LIN {X 0,Y 404.076,Z 442.331,A -85,B 0,C 180,E1 -11324.748,E2 -11324.748} C_VEL
LIN {X 0,Y 402.953,Z 452.471,A -85,B 0,C 180,E1 -11326.125,E2 -11326.125} C_VEL
LIN {X 0,Y 401.871,Z 461.516,A -85,B 0,C 180,E1 -11327.63,E2 -11327.63} C_VEL
LIN {X 0,Y 400.856,Z 469.336,A -85,B 0,C 180,E1 -11329.213,E2 -11329.213} C_VEL
LIN {X 0,Y 399.877,Z 476.001,A -85,B 0,C 180,E1 -11330.899,E2 -11330.899} C_VEL
LIN {X 0,Y 399.254,Z 480.643,A -85,B 0,C 180,E1 -11332.414,E2 -11332.414} C_VEL
LIN {X 0,Y 398.694,Z 484.232,A -85,B 0,C 180,E1 -11333.929,E2 -11333.929} C_VEL
LIN {X 0,Y 398.541,Z 486.049,A -85,B 0,C 180,E1 -11334.942,E2 -11334.942} C_VEL
LIN {X 0,Y 398.272,Z 487.43,A -85,B 0,C 180,E1 -11335.953,E2 -11335.953} C_VEL
LIN {X 0,Y 398.06,Z 488.39,A -85,B 0,C 180,E1 -11336.964,E2 -11336.964} C_VEL
LIN {X 0,Y 397.79,Z 488.969,A -85,B 0,C 180,E1 -11337.975,E2 -11337.975} C_VEL
LIN {X 0,Y 397.658,Z 489.133,A -85,B 0,C 180,E1 -11338.988,E2 -11338.988} C_VEL
LIN {X 0,Y 397.526,Z 488.893,A -85,B 0,C 180,E1 -11340,E2 -11340} C_VEL
LIN {X 0,Y 397.495,Z 488.205,A -85,B 0,C 180,E1 -11341.013,E2 -11341.013} C_VEL
LIN {X 0,Y 397.414,Z 487.123,A -85,B 0,C 180,E1 -11342.027,E2 -11342.027} C_VEL
LIN {X 0,Y 397.512,Z 485.612,A -85,B 0,C 180,E1 -11343.041,E2 -11343.041} C_VEL
LIN {X 0,Y 397.477,Z 482.566,A -85,B 0,C 180,E1 -11344.564,E2 -11344.564} C_VEL
LIN {X 0,Y 397.578,Z 478.489,A -85,B 0,C 180,E1 -11346.089,E2 -11346.089} C_VEL
LIN {X 0,Y 398.065,Z 473.274,A -85,B 0,C 180,E1 -11347.61,E2 -11347.61} C_VEL
LIN {X 0,Y 398.488,Z 465.684,A -85,B 0,C 180,E1 -11349.39,E2 -11349.39} C_VEL
LIN {X 0,Y 398.962,Z 457.56,A -85,B 0,C 180,E1 -11350.916,E2 -11350.916} C_VEL
LIN {X 0,Y 399.517,Z 447.676,A -85,B 0,C 180,E1 -11352.445,E2 -11352.445} C_VEL
LIN {X 0,Y 400.278,Z 437.712,A -85,B 0,C 180,E1 -11353.712,E2 -11353.712} C_VEL
LIN {X 0,Y 400.99,Z 425.569,A -85,B 0,C 180,E1 -11354.983,E2 -11354.983} C_VEL
LIN {X 0,Y 401.633,Z 413.729,A -85,B 0,C 180,E1 -11355.995,E2 -11355.995} C_VEL
LIN {X 0,Y 402.443,Z 400.813,A -85,B 0,C 180,E1 -11356.878,E2 -11356.878} C_VEL
LIN {X 0,Y 402.734,Z 392.913,A -85,B 0,C 180,E1 -11357.323,E2 -11357.323} C_VEL
LIN {X 0,Y 399.412,Z 378.284,A -85,B 0,C 180,E1 -11358.158,E2 -11358.158} C_VEL
LIN {X 0,Y 396.905,Z 368.546,A -85,B 0,C 180,E1 -11358.62,E2 -11358.62} C_VEL
LIN {X 0,Y 397.081,Z 362.565,A -85,B 0,C 180,E1 -11361.82,E2 -11361.82} C_VEL
LIN {X 0,Y 397.308,Z 355.709,A -85,B 0,C 180,E1 -11365.556,E2 -11365.556} C_VEL
LIN {X 0,Y 397.543,Z 349.381,A -85,B 0,C 180,E1 -11369.089,E2 -11369.089} C_VEL
LIN {X 0,Y 397.831,Z 343.175,A -85,B 0,C 180,E1 -11372.603,E2 -11372.603} C_VEL
LIN {X 0,Y 397.935,Z 337.889,A -85,B 0,C 180,E1 -11375.665,E2 -11375.665} C_VEL
LIN {X 0,Y 397.733,Z 335.123,A -85,B 0,C 180,E1 -11377.328,E2 -11377.328} C_VEL
LIN {X 0,Y 397.121,Z 331.336,A -85,B 0,C 180,E1 -11379.735,E2 -11379.735} C_VEL
LIN {X 0,Y 397.109,Z 331.334,A -85,B 0,C 180,E1 -11383.648,E2 -11383.648} C_VEL
LIN {X 0,Y 397.11,Z 331.332,A -85,B 0,C 180,E1 -11386.52,E2 -11386.52} C_VEL
LIN {X 0,Y 397.128,Z 331.421,A -85,B 0,C 180,E1 -11390.027,E2 -11390.027} C_VEL
LIN {X 0,Y 398.424,Z 338.477,A -85,B 0,C 180,E1 -11393.146,E2 -11393.146} C_VEL
LIN {X 0,Y 398.848,Z 342.731,A -85,B 0,C 180,E1 -11395.061,E2 -11395.061} C_VEL
LIN {X 0,Y 398.687,Z 350.568,A -85,B 0,C 180,E1 -11398.664,E2 -11398.664} C_VEL
LIN {X 0,Y 398.55,Z 357.361,A -85,B 0,C 180,E1 -11401.848,E2 -11401.848} C_VEL
LIN {X 0,Y 398.521,Z 365.236,A -85,B 0,C 180,E1 -11405.515,E2 -11405.515} C_VEL
LIN {X 0,Y 398.622,Z 373.552,A -85,B 0,C 180,E1 -11409.137,E2 -11409.137} C_VEL
LIN {X 0,Y 398.818,Z 380.793,A -85,B 0,C 180,E1 -11411.941,E2 -11411.941} C_VEL
LIN {X 0,Y 402.682,Z 393.199,A -85,B 0,C 180,E1 -11412.494,E2 -11412.494} C_VEL
LIN {X 0,Y 403.209,Z 396.027,A -85,B 0,C 180,E1 -11412.631,E2 -11412.631} C_VEL
LIN {X 0,Y 402.908,Z 408.015,A -85,B 0,C 180,E1 -11413.206,E2 -11413.206} C_VEL
LIN {X 0,Y 402.433,Z 419.434,A -85,B 0,C 180,E1 -11413.95,E2 -11413.95} C_VEL
LIN {X 0,Y 401.82,Z 430.918,A -85,B 0,C 180,E1 -11414.918,E2 -11414.918} C_VEL
LIN {X 0,Y 401.129,Z 441.593,A -85,B 0,C 180,E1 -11416.058,E2 -11416.058} C_VEL
LIN {X 0,Y 400.428,Z 451.077,A -85,B 0,C 180,E1 -11417.325,E2 -11417.325} C_VEL
LIN {X 0,Y 399.552,Z 460.293,A -85,B 0,C 180,E1 -11418.841,E2 -11418.841} C_VEL
LIN {X 0,Y 398.974,Z 467.575,A -85,B 0,C 180,E1 -11420.365,E2 -11420.365} C_VEL
LIN {X 0,Y 398.52,Z 473.405,A -85,B 0,C 180,E1 -11421.887,E2 -11421.887} C_VEL
LIN {X 0,Y 397.835,Z 478.062,A -85,B 0,C 180,E1 -11423.404,E2 -11423.404} C_VEL
LIN {X 0,Y 397.571,Z 481.583,A -85,B 0,C 180,E1 -11424.927,E2 -11424.927} C_VEL
LIN {X 0,Y 397.535,Z 483.38,A -85,B 0,C 180,E1 -11425.943,E2 -11425.943} C_VEL
LIN {X 0,Y 397.447,Z 484.762,A -85,B 0,C 180,E1 -11426.957,E2 -11426.957} C_VEL
LIN {X 0,Y 397.196,Z 486.352,A -85,B 0,C 180,E1 -11428.984,E2 -11428.984} C_VEL
LIN {X 0,Y 397.16,Z 486.586,A -85,B 0,C 180,E1 -11429.998,E2 -11429.998} C_VEL
LIN {X 0,Y 397.293,Z 485.82,A -85,B 0,C 180,E1 -11432.025,E2 -11432.025} C_VEL
LIN {X 0,Y 397.459,Z 484.866,A -85,B 0,C 180,E1 -11433.038,E2 -11433.038} C_VEL
LIN {X 0,Y 397.552,Z 483.541,A -85,B 0,C 180,E1 -11434.052,E2 -11434.052} C_VEL
LIN {X 0,Y 397.722,Z 480.756,A -85,B 0,C 180,E1 -11435.575,E2 -11435.575} C_VEL
LIN {X 0,Y 398.1,Z 476.945,A -85,B 0,C 180,E1 -11437.096,E2 -11437.096} C_VEL
LIN {X 0,Y 398.64,Z 471.995,A -85,B 0,C 180,E1 -11438.616,E2 -11438.616} C_VEL
LIN {X 0,Y 398.848,Z 469.563,A -85,B 0,C 180,E1 -11439.249,E2 -11439.249} C_VEL
LIN {X 0,Y 398.363,Z 467.668,A -85,B 0,C 180,E1 -11439.75,E2 -11439.75} C_VEL
LIN {X 0,Y 393.286,Z 461.707,A -85,B 0,C 180,E1 -11441.349,E2 -11441.349} C_VEL
LIN {X 0,Y 392.936,Z 459.353,A -85,B 0,C 180,E1 -11441.816,E2 -11441.816} C_VEL
LIN {X 0,Y 393.736,Z 451.114,A -85,B 0,C 180,E1 -11443.152,E2 -11443.152} C_VEL
LIN {X 0,Y 394.369,Z 442.445,A -85,B 0,C 180,E1 -11444.313,E2 -11444.313} C_VEL
LIN {X 0,Y 395.042,Z 431.694,A -85,B 0,C 180,E1 -11445.474,E2 -11445.474} C_VEL
LIN {X 0,Y 395.736,Z 420.066,A -85,B 0,C 180,E1 -11446.462,E2 -11446.462} C_VEL
LIN {X 0,Y 396.267,Z 408.557,A -85,B 0,C 180,E1 -11447.212,E2 -11447.212} C_VEL
LIN {X 0,Y 396.362,Z 396.075,A -85,B 0,C 180,E1 -11447.817,E2 -11447.817} C_VEL
LIN {X 0,Y 392.761,Z 384.449,A -85,B 0,C 180,E1 -11448.381,E2 -11448.381} C_VEL
LIN {X 0,Y 391.906,Z 381.637,A -85,B 0,C 180,E1 -11448.505,E2 -11448.505} C_VEL
LIN {X 0,Y 391.687,Z 373.901,A -85,B 0,C 180,E1 -11451.578,E2 -11451.578} C_VEL
LIN {X 0,Y 391.648,Z 367.501,A -85,B 0,C 180,E1 -11454.373,E2 -11454.373} C_VEL
LIN {X 0,Y 391.635,Z 359.97,A -85,B 0,C 180,E1 -11457.809,E2 -11457.809} C_VEL
LIN {X 0,Y 391.769,Z 354.179,A -85,B 0,C 180,E1 -11460.561,E2 -11460.561} C_VEL
LIN {X 0,Y 391.906,Z 347.231,A -85,B 0,C 180,E1 -11463.77,E2 -11463.77} C_VEL
LIN {X 0,Y 391.796,Z 341.719,A -85,B 0,C 180,E1 -11466.292,E2 -11466.292} C_VEL
LIN {X 0,Y 390.605,Z 335.016,A -85,B 0,C 180,E1 -11469.314,E2 -11469.314} C_VEL
LIN {X 0,Y 390.047,Z 332.214,A -85,B 0,C 180,E1 -11470.531,E2 -11470.531} C_VEL
LIN {X 0,Y 390.044,Z 332.214,A -85,B 0,C 180,E1 -11473.884,E2 -11473.884} C_VEL
LIN {X 0,Y 390.099,Z 332.208,A -85,B 0,C 180,E1 -11476.795,E2 -11476.795} C_VEL
LIN {X 0,Y 390.063,Z 332.208,A -85,B 0,C 180,E1 -11479.561,E2 -11479.561} C_VEL
LIN {X 0,Y 390.031,Z 332.215,A -85,B 0,C 180,E1 -11482.446,E2 -11482.446} C_VEL
LIN {X 0,Y 390.05,Z 332.211,A -85,B 0,C 180,E1 -11486.043,E2 -11486.043} C_VEL
LIN {X 0,Y 390.027,Z 332.209,A -85,B 0,C 180,E1 -11489.867,E2 -11489.867} C_VEL
LIN {X 0,Y 390.093,Z 332.199,A -85,B 0,C 180,E1 -11493.23,E2 -11493.23} C_VEL
LIN {X 0,Y 390.102,Z 332.198,A -85,B 0,C 180,E1 -11496.743,E2 -11496.743} C_VEL
LIN {X 0,Y 390.108,Z 332.202,A -85,B 0,C 180,E1 -11499.983,E2 -11499.983} C_VEL
LIN {X 0,Y 390.115,Z 332.206,A -85,B 0,C 180,E1 -11503.247,E2 -11503.247} C_VEL
LIN {X 0,Y 390.171,Z 332.189,A -85,B 0,C 180,E1 -11506.56,E2 -11506.56} C_VEL
LIN {X 0,Y 390.159,Z 332.195,A -85,B 0,C 180,E1 -11509.622,E2 -11509.622} C_VEL
LIN {X 0,Y 390.294,Z 332.18,A -85,B 0,C 180,E1 -11512.758,E2 -11512.758} C_VEL
LIN {X 0,Y 390.203,Z 332.187,A -85,B 0,C 180,E1 -11514.833,E2 -11514.833} C_VEL
LIN {X 0,Y 390.392,Z 332.168,A -85,B 0,C 180,E1 -11517.936,E2 -11517.936} C_VEL
LIN {X 0,Y 390.524,Z 332.147,A -85,B 0,C 180,E1 -11520,E2 -11520} C_VEL
LIN {X 0,Y 390.328,Z 332.176,A -85,B 0,C 180,E1 -11523.096,E2 -11523.096} C_VEL
LIN {X 0,Y 390.317,Z 332.177,A -85,B 0,C 180,E1 -11526.202,E2 -11526.202} C_VEL
LIN {X 0,Y 390.29,Z 332.181,A -85,B 0,C 180,E1 -11528.282,E2 -11528.282} C_VEL
LIN {X 0,Y 390.154,Z 332.2,A -85,B 0,C 180,E1 -11532.483,E2 -11532.483} C_VEL
LIN {X 0,Y 390.12,Z 332.202,A -85,B 0,C 180,E1 -11535.677,E2 -11535.677} C_VEL
LIN {X 0,Y 390.097,Z 332.205,A -85,B 0,C 180,E1 -11538.922,E2 -11538.922} C_VEL
LIN {X 0,Y 390.09,Z 332.206,A -85,B 0,C 180,E1 -11542.231,E2 -11542.231} C_VEL
LIN {X 0,Y 390.096,Z 332.204,A -85,B 0,C 180,E1 -11545.745,E2 -11545.745} C_VEL
LIN {X 0,Y 390.036,Z 332.212,A -85,B 0,C 180,E1 -11549.111,E2 -11549.111} C_VEL
LIN {X 0,Y 390.021,Z 332.216,A -85,B 0,C 180,E1 -11552.723,E2 -11552.723} C_VEL
LIN {X 0,Y 390.037,Z 332.214,A -85,B 0,C 180,E1 -11555.827,E2 -11555.827} C_VEL
LIN {X 0,Y 390.027,Z 332.217,A -85,B 0,C 180,E1 -11557.466,E2 -11557.466} C_VEL
LIN {X 0,Y 392.821,Z 341.775,A -85,B 0,C 180,E1 -11560.77,E2 -11560.77} C_VEL
LIN {X 0,Y 395.179,Z 349.812,A -85,B 0,C 180,E1 -11563.359,E2 -11563.359} C_VEL
LIN {X 0,Y 398.223,Z 359.679,A -85,B 0,C 180,E1 -11566.351,E2 -11566.351} C_VEL
LIN {X 0,Y 401.682,Z 372.211,A -85,B 0,C 180,E1 -11569.826,E2 -11569.826} C_VEL
LIN {X 0,Y 403.335,Z 378.619,A -85,B 0,C 180,E1 -11571.49,E2 -11571.49} C_VEL
LIN {X 0,Y 401.079,Z 392.2,A -85,B 0,C 180,E1 -11574.368,E2 -11574.368} C_VEL
LIN {X 0,Y 398.451,Z 410.185,A -85,B 0,C 180,E1 -11578.056,E2 -11578.056} C_VEL
LIN {X 0,Y 397.562,Z 416.992,A -85,B 0,C 180,E1 -11579.407,E2 -11579.407} C_VEL
LIN {X 0,Y 401.91,Z 440.861,A -85,B 0,C 180,E1 -11580.3,E2 -11580.3} C_VEL
LIN {X 0,Y 404.613,Z 456.32,A -85,B 0,C 180,E1 -11581.044,E2 -11581.044} C_VEL
LIN {X 0,Y 404.439,Z 460.912,A -85,B 0,C 180,E1 -11581.246,E2 -11581.246} C_VEL
LIN {X 0,Y 403.168,Z 476.373,A -85,B 0,C 180,E1 -11581.997,E2 -11581.997} C_VEL
LIN {X 0,Y 401.594,Z 491.749,A -85,B 0,C 180,E1 -11582.938,E2 -11582.938} C_VEL
LIN {X 0,Y 399.977,Z 506.825,A -85,B 0,C 180,E1 -11584.086,E2 -11584.086} C_VEL
LIN {X 0,Y 398.034,Z 521.978,A -85,B 0,C 180,E1 -11585.488,E2 -11585.488} C_VEL
LIN {X 0,Y 396.209,Z 535.794,A -85,B 0,C 180,E1 -11587.034,E2 -11587.034} C_VEL
LIN {X 0,Y 394.645,Z 547.575,A -85,B 0,C 180,E1 -11588.591,E2 -11588.591} C_VEL
LIN {X 0,Y 393.104,Z 559.357,A -85,B 0,C 180,E1 -11590.417,E2 -11590.417} C_VEL
LIN {X 0,Y 391.862,Z 569.445,A -85,B 0,C 180,E1 -11592.251,E2 -11592.251} C_VEL
LIN {X 0,Y 390.905,Z 578.006,A -85,B 0,C 180,E1 -11594.09,E2 -11594.09} C_VEL
LIN {X 0,Y 390.138,Z 585.358,A -85,B 0,C 180,E1 -11595.928,E2 -11595.928} C_VEL
LIN {X 0,Y 389.592,Z 592.418,A -85,B 0,C 180,E1 -11598.03,E2 -11598.03} C_VEL
LIN {X 0,Y 389.136,Z 599.389,A -85,B 0,C 180,E1 -11600.648,E2 -11600.648} C_VEL
LIN {X 0,Y 389.044,Z 603.593,A -85,B 0,C 180,E1 -11602.738,E2 -11602.738} C_VEL
LIN {X 0,Y 388.924,Z 606.727,A -85,B 0,C 180,E1 -11604.819,E2 -11604.819} C_VEL
LIN {X 0,Y 389.013,Z 608.747,A -85,B 0,C 180,E1 -11606.896,E2 -11606.896} C_VEL
LIN {X 0,Y 388.938,Z 609.723,A -85,B 0,C 180,E1 -11608.967,E2 -11608.967} C_VEL
LIN {X 0,Y 388.95,Z 609.638,A -85,B 0,C 180,E1 -11611.038,E2 -11611.038} C_VEL
LIN {X 0,Y 389.015,Z 608.518,A -85,B 0,C 180,E1 -11613.109,E2 -11613.109} C_VEL
LIN {X 0,Y 388.996,Z 606.322,A -85,B 0,C 180,E1 -11615.185,E2 -11615.185} C_VEL
LIN {X 0,Y 389.116,Z 603.015,A -85,B 0,C 180,E1 -11617.266,E2 -11617.266} C_VEL
LIN {X 0,Y 389.18,Z 598.597,A -85,B 0,C 180,E1 -11619.356,E2 -11619.356} C_VEL
LIN {X 0,Y 389.517,Z 592.896,A -85,B 0,C 180,E1 -11621.45,E2 -11621.45} C_VEL
LIN {X 0,Y 390.058,Z 585.925,A -85,B 0,C 180,E1 -11623.549,E2 -11623.549} C_VEL
LIN {X 0,Y 390.776,Z 577.523,A -85,B 0,C 180,E1 -11625.653,E2 -11625.653} C_VEL
LIN {X 0,Y 391.728,Z 568.779,A -85,B 0,C 180,E1 -11627.491,E2 -11627.491} C_VEL
LIN {X 0,Y 392.86,Z 558.606,A -85,B 0,C 180,E1 -11629.329,E2 -11629.329} C_VEL
LIN {X 0,Y 394.283,Z 546.745,A -85,B 0,C 180,E1 -11631.161,E2 -11631.161} C_VEL
LIN {X 0,Y 395.884,Z 534.224,A -85,B 0,C 180,E1 -11632.81,E2 -11632.81} C_VEL
LIN {X 0,Y 397.661,Z 519.904,A -85,B 0,C 180,E1 -11634.403,E2 -11634.403} C_VEL
LIN {X 0,Y 399.568,Z 504.73,A -85,B 0,C 180,E1 -11635.808,E2 -11635.808} C_VEL
LIN {X 0,Y 401.236,Z 489.324,A -85,B 0,C 180,E1 -11636.993,E2 -11636.993} C_VEL
LIN {X 0,Y 402.885,Z 473.844,A -85,B 0,C 180,E1 -11637.959,E2 -11637.959} C_VEL
LIN {X 0,Y 404.326,Z 456.774,A -85,B 0,C 180,E1 -11638.808,E2 -11638.808} C_VEL
LIN {X 0,Y 401.862,Z 440.786,A -85,B 0,C 180,E1 -11639.681,E2 -11639.681} C_VEL
LIN {X 0,Y 399.853,Z 426.098,A -85,B 0,C 180,E1 -11640.329,E2 -11640.329} C_VEL
LIN {X 0,Y 397.477,Z 414.254,A -85,B 0,C 180,E1 -11640.887,E2 -11640.887} C_VEL
LIN {X 0,Y 400.109,Z 398.368,A -85,B 0,C 180,E1 -11644.355,E2 -11644.355} C_VEL
LIN {X 0,Y 402.972,Z 386.243,A -85,B 0,C 180,E1 -11647.306,E2 -11647.306} C_VEL
LIN {X 0,Y 404.249,Z 381.682,A -85,B 0,C 180,E1 -11648.525,E2 -11648.525} C_VEL
LIN {X 0,Y 404.093,Z 379.075,A -85,B 0,C 180,E1 -11649.408,E2 -11649.408} C_VEL
LIN {X 0,Y 402.704,Z 374.043,A -85,B 0,C 180,E1 -11651.545,E2 -11651.545} C_VEL
LIN {X 0,Y 401.865,Z 371.224,A -85,B 0,C 180,E1 -11653.006,E2 -11653.006} C_VEL
LIN {X 0,Y 400.572,Z 367.722,A -85,B 0,C 180,E1 -11655.429,E2 -11655.429} C_VEL
LIN {X 0,Y 399.586,Z 365.374,A -85,B 0,C 180,E1 -11658.061,E2 -11658.061} C_VEL
LIN {X 0,Y 398.795,Z 364.51,A -85,B 0,C 180,E1 -11660.623,E2 -11660.623} C_VEL
LIN {X 0,Y 398.072,Z 364.839,A -85,B 0,C 180,E1 -11663.111,E2 -11663.111} C_VEL
LIN {X 0,Y 397.049,Z 366.226,A -85,B 0,C 180,E1 -11665.5,E2 -11665.5} C_VEL
LIN {X 0,Y 395.551,Z 369.392,A -85,B 0,C 180,E1 -11668.986,E2 -11668.986} C_VEL
LIN {X 0,Y 394.433,Z 373.268,A -85,B 0,C 180,E1 -11672.402,E2 -11672.402} C_VEL
LIN {X 0,Y 393.72,Z 377.587,A -85,B 0,C 180,E1 -11675.761,E2 -11675.761} C_VEL
LIN {X 0,Y 393.268,Z 381.308,A -85,B 0,C 180,E1 -11678.326,E2 -11678.326} C_VEL
LIN {X 0,Y 399.181,Z 395.499,A -85,B 0,C 180,E1 -11679.827,E2 -11679.827} C_VEL
LIN {X 0,Y 401.993,Z 404.636,A -85,B 0,C 180,E1 -11680.751,E2 -11680.751} C_VEL
LIN {X 0,Y 400.446,Z 419.286,A -85,B 0,C 180,E1 -11681.844,E2 -11681.844} C_VEL
LIN {X 0,Y 398.954,Z 432.684,A -85,B 0,C 180,E1 -11683.103,E2 -11683.103} C_VEL
LIN {X 0,Y 397.652,Z 443.666,A -85,B 0,C 180,E1 -11684.364,E2 -11684.364} C_VEL
LIN {X 0,Y 396.316,Z 454.53,A -85,B 0,C 180,E1 -11685.888,E2 -11685.888} C_VEL
LIN {X 0,Y 395.187,Z 463.434,A -85,B 0,C 180,E1 -11687.417,E2 -11687.417} C_VEL
LIN {X 0,Y 394.132,Z 470.792,A -85,B 0,C 180,E1 -11688.958,E2 -11688.958} C_VEL
LIN {X 0,Y 393.073,Z 477.647,A -85,B 0,C 180,E1 -11690.74,E2 -11690.74} C_VEL
LIN {X 0,Y 392.402,Z 482.213,A -85,B 0,C 180,E1 -11692.281,E2 -11692.281} C_VEL
LIN {X 0,Y 391.799,Z 485.706,A -85,B 0,C 180,E1 -11693.822,E2 -11693.822} C_VEL
LIN {X 0,Y 391.627,Z 487.463,A -85,B 0,C 180,E1 -11694.852,E2 -11694.852} C_VEL
LIN {X 0,Y 391.331,Z 488.805,A -85,B 0,C 180,E1 -11695.881,E2 -11695.881} C_VEL
LIN {X 0,Y 391.113,Z 489.728,A -85,B 0,C 180,E1 -11696.91,E2 -11696.91} C_VEL
LIN {X 0,Y 390.836,Z 490.269,A -85,B 0,C 180,E1 -11697.939,E2 -11697.939} C_VEL
LIN {X 0,Y 390.695,Z 490.391,A -85,B 0,C 180,E1 -11698.97,E2 -11698.97} C_VEL
LIN {X 0,Y 390.547,Z 490.095,A -85,B 0,C 180,E1 -11700,E2 -11700} C_VEL
LIN {X 0,Y 390.501,Z 489.359,A -85,B 0,C 180,E1 -11701.032,E2 -11701.032} C_VEL
LIN {X 0,Y 390.428,Z 488.234,A -85,B 0,C 180,E1 -11702.064,E2 -11702.064} C_VEL
LIN {X 0,Y 390.505,Z 486.689,A -85,B 0,C 180,E1 -11703.095,E2 -11703.095} C_VEL
LIN {X 0,Y 390.471,Z 483.564,A -85,B 0,C 180,E1 -11704.646,E2 -11704.646} C_VEL
LIN {X 0,Y 390.594,Z 479.411,A -85,B 0,C 180,E1 -11706.198,E2 -11706.198} C_VEL
LIN {X 0,Y 391.081,Z 474.119,A -85,B 0,C 180,E1 -11707.746,E2 -11707.746} C_VEL
LIN {X 0,Y 391.543,Z 466.408,A -85,B 0,C 180,E1 -11709.558,E2 -11709.558} C_VEL
LIN {X 0,Y 392.037,Z 458.194,A -85,B 0,C 180,E1 -11711.112,E2 -11711.112} C_VEL
LIN {X 0,Y 392.628,Z 448.224,A -85,B 0,C 180,E1 -11712.667,E2 -11712.667} C_VEL
LIN {X 0,Y 393.489,Z 437.028,A -85,B 0,C 180,E1 -11714.085,E2 -11714.085} C_VEL
LIN {X 0,Y 394.229,Z 424.58,A -85,B 0,C 180,E1 -11715.378,E2 -11715.378} C_VEL
LIN {X 0,Y 394.927,Z 412.444,A -85,B 0,C 180,E1 -11716.401,E2 -11716.401} C_VEL
LIN {X 0,Y 395.697,Z 398.852,A -85,B 0,C 180,E1 -11717.308,E2 -11717.308} C_VEL
LIN {X 0,Y 395.771,Z 393.106,A -85,B 0,C 180,E1 -11717.637,E2 -11717.637} C_VEL
LIN {X 0,Y 392.444,Z 378.929,A -85,B 0,C 180,E1 -11718.465,E2 -11718.465} C_VEL
LIN {X 0,Y 389.864,Z 368.891,A -85,B 0,C 180,E1 -11718.969,E2 -11718.969} C_VEL
LIN {X 0,Y 390.087,Z 362.868,A -85,B 0,C 180,E1 -11722.232,E2 -11722.232} C_VEL
LIN {X 0,Y 390.301,Z 356.38,A -85,B 0,C 180,E1 -11725.795,E2 -11725.795} C_VEL
LIN {X 0,Y 390.544,Z 350.55,A -85,B 0,C 180,E1 -11729.07,E2 -11729.07} C_VEL
LIN {X 0,Y 390.849,Z 344.32,A -85,B 0,C 180,E1 -11732.646,E2 -11732.646} C_VEL
LIN {X 0,Y 390.967,Z 340.088,A -85,B 0,C 180,E1 -11735.116,E2 -11735.116} C_VEL
LIN {X 0,Y 390.811,Z 336.913,A -85,B 0,C 180,E1 -11737.022,E2 -11737.022} C_VEL
LIN {X 0,Y 390.083,Z 332.212,A -85,B 0,C 180,E1 -11739.958,E2 -11739.958} C_VEL
LIN {X 0,Y 390.063,Z 332.212,A -85,B 0,C 180,E1 -11743.885,E2 -11743.885} C_VEL
LIN {X 0,Y 390.065,Z 332.21,A -85,B 0,C 180,E1 -11746.788,E2 -11746.788} C_VEL
LIN {X 0,Y 390.077,Z 332.33,A -85,B 0,C 180,E1 -11749.637,E2 -11749.637} C_VEL
LIN {X 0,Y 391.26,Z 338.426,A -85,B 0,C 180,E1 -11752.356,E2 -11752.356} C_VEL
LIN {X 0,Y 391.929,Z 342.986,A -85,B 0,C 180,E1 -11754.415,E2 -11754.415} C_VEL
LIN {X 0,Y 391.812,Z 349.656,A -85,B 0,C 180,E1 -11757.464,E2 -11757.464} C_VEL
LIN {X 0,Y 391.663,Z 357.249,A -85,B 0,C 180,E1 -11761.019,E2 -11761.019} C_VEL
LIN {X 0,Y 391.57,Z 364.696,A -85,B 0,C 180,E1 -11764.482,E2 -11764.482} C_VEL
LIN {X 0,Y 391.684,Z 372.316,A -85,B 0,C 180,E1 -11767.862,E2 -11767.862} C_VEL
LIN {X 0,Y 391.891,Z 381.376,A -85,B 0,C 180,E1 -11771.507,E2 -11771.507} C_VEL
LIN {X 0,Y 391.943,Z 381.903,A -85,B 0,C 180,E1 -11771.615,E2 -11771.615} C_VEL
LIN {X 0,Y 395.741,Z 394.002,A -85,B 0,C 180,E1 -11772.166,E2 -11772.166} C_VEL
LIN {X 0,Y 396.497,Z 397.068,A -85,B 0,C 180,E1 -11772.327,E2 -11772.327} C_VEL
LIN {X 0,Y 396.198,Z 409.069,A -85,B 0,C 180,E1 -11772.912,E2 -11772.912} C_VEL
LIN {X 0,Y 395.692,Z 420.473,A -85,B 0,C 180,E1 -11773.667,E2 -11773.667} C_VEL
LIN {X 0,Y 395.047,Z 431.985,A -85,B 0,C 180,E1 -11774.653,E2 -11774.653} C_VEL
LIN {X 0,Y 394.327,Z 442.663,A -85,B 0,C 180,E1 -11775.812,E2 -11775.812} C_VEL
LIN {X 0,Y 393.586,Z 452.15,A -85,B 0,C 180,E1 -11777.1,E2 -11777.1} C_VEL
LIN {X 0,Y 392.67,Z 461.368,A -85,B 0,C 180,E1 -11778.643,E2 -11778.643} C_VEL
LIN {X 0,Y 392.057,Z 468.651,A -85,B 0,C 180,E1 -11780.193,E2 -11780.193} C_VEL
LIN {X 0,Y 391.586,Z 474.479,A -85,B 0,C 180,E1 -11781.743,E2 -11781.743} C_VEL
LIN {X 0,Y 390.865,Z 479.139,A -85,B 0,C 180,E1 -11783.286,E2 -11783.286} C_VEL
LIN {X 0,Y 390.582,Z 482.66,A -85,B 0,C 180,E1 -11784.836,E2 -11784.836} C_VEL
LIN {X 0,Y 390.535,Z 484.457,A -85,B 0,C 180,E1 -11785.87,E2 -11785.87} C_VEL
LIN {X 0,Y 390.449,Z 485.838,A -85,B 0,C 180,E1 -11786.902,E2 -11786.902} C_VEL
LIN {X 0,Y 390.18,Z 487.429,A -85,B 0,C 180,E1 -11788.965,E2 -11788.965} C_VEL
LIN {X 0,Y 390.143,Z 487.662,A -85,B 0,C 180,E1 -11789.997,E2 -11789.997} C_VEL
LIN {X 0,Y 390.283,Z 486.896,A -85,B 0,C 180,E1 -11792.061,E2 -11792.061} C_VEL
LIN {X 0,Y 390.46,Z 485.94,A -85,B 0,C 180,E1 -11793.093,E2 -11793.093} C_VEL
LIN {X 0,Y 390.55,Z 484.617,A -85,B 0,C 180,E1 -11794.125,E2 -11794.125} C_VEL
LIN {X 0,Y 390.735,Z 481.831,A -85,B 0,C 180,E1 -11795.675,E2 -11795.675} C_VEL
LIN {X 0,Y 391.14,Z 478.019,A -85,B 0,C 180,E1 -11797.223,E2 -11797.223} C_VEL
LIN {X 0,Y 391.721,Z 473.065,A -85,B 0,C 180,E1 -11798.769,E2 -11798.769} C_VEL
LIN {X 0,Y 392.235,Z 466.839,A -85,B 0,C 180,E1 -11800.319,E2 -11800.319} C_VEL
LIN {X 0,Y 392.936,Z 459.353,A -85,B 0,C 180,E1 -11801.816,E2 -11801.816} C_VEL
LIN {X 0,Y 392.795,Z 455.651,A -85,B 0,C 180,E1 -11802.485,E2 -11802.485} C_VEL
LIN {X 0,Y 390.635,Z 449.529,A -85,B 0,C 180,E1 -11803.582,E2 -11803.582} C_VEL
LIN {X 0,Y 388.331,Z 442.875,A -85,B 0,C 180,E1 -11804.612,E2 -11804.612} C_VEL
LIN {X 0,Y 387.957,Z 438.338,A -85,B 0,C 180,E1 -11805.169,E2 -11805.169} C_VEL
LIN {X 0,Y 388.629,Z 429.221,A -85,B 0,C 180,E1 -11806.079,E2 -11806.079} C_VEL
LIN {X 0,Y 389.194,Z 416.864,A -85,B 0,C 180,E1 -11807.061,E2 -11807.061} C_VEL
LIN {X 0,Y 389.723,Z 404.702,A -85,B 0,C 180,E1 -11807.782,E2 -11807.782} C_VEL
LIN {X 0,Y 389.632,Z 397.339,A -85,B 0,C 180,E1 -11808.126,E2 -11808.126} C_VEL
LIN {X 0,Y 385.706,Z 384.719,A -85,B 0,C 180,E1 -11808.749,E2 -11808.749} C_VEL
LIN {X 0,Y 384.998,Z 382.579,A -85,B 0,C 180,E1 -11808.871,E2 -11808.871} C_VEL
LIN {X 0,Y 384.818,Z 374.751,A -85,B 0,C 180,E1 -11811.984,E2 -11811.984} C_VEL
LIN {X 0,Y 384.752,Z 368.209,A -85,B 0,C 180,E1 -11814.839,E2 -11814.839} C_VEL
LIN {X 0,Y 384.79,Z 359.677,A -85,B 0,C 180,E1 -11818.753,E2 -11818.753} C_VEL
LIN {X 0,Y 384.916,Z 352.881,A -85,B 0,C 180,E1 -11821.968,E2 -11821.968} C_VEL
LIN {X 0,Y 385.055,Z 345.889,A -85,B 0,C 180,E1 -11825.185,E2 -11825.185} C_VEL
LIN {X 0,Y 384.663,Z 341.762,A -85,B 0,C 180,E1 -11827.076,E2 -11827.076} C_VEL
LIN {X 0,Y 383.475,Z 335.526,A -85,B 0,C 180,E1 -11829.896,E2 -11829.896} C_VEL
LIN {X 0,Y 382.983,Z 333.093,A -85,B 0,C 180,E1 -11831.001,E2 -11831.001} C_VEL
LIN {X 0,Y 382.993,Z 333.09,A -85,B 0,C 180,E1 -11834.302,E2 -11834.302} C_VEL
LIN {X 0,Y 383.06,Z 333.082,A -85,B 0,C 180,E1 -11837.246,E2 -11837.246} C_VEL
LIN {X 0,Y 383.007,Z 333.09,A -85,B 0,C 180,E1 -11840.409,E2 -11840.409} C_VEL
LIN {X 0,Y 383.009,Z 333.086,A -85,B 0,C 180,E1 -11844.042,E2 -11844.042} C_VEL
LIN {X 0,Y 382.968,Z 333.093,A -85,B 0,C 180,E1 -11847.576,E2 -11847.576} C_VEL
LIN {X 0,Y 382.972,Z 333.087,A -85,B 0,C 180,E1 -11850.298,E2 -11850.298} C_VEL
LIN {X 0,Y 383.06,Z 333.076,A -85,B 0,C 180,E1 -11854.019,E2 -11854.019} C_VEL
LIN {X 0,Y 383.036,Z 333.077,A -85,B 0,C 180,E1 -11857.337,E2 -11857.337} C_VEL
LIN {X 0,Y 383.055,Z 333.079,A -85,B 0,C 180,E1 -11860.716,E2 -11860.716} C_VEL
LIN {X 0,Y 383.058,Z 333.081,A -85,B 0,C 180,E1 -11864.025,E2 -11864.025} C_VEL
LIN {X 0,Y 383.12,Z 333.073,A -85,B 0,C 180,E1 -11867.283,E2 -11867.283} C_VEL
LIN {X 0,Y 383.135,Z 333.063,A -85,B 0,C 180,E1 -11870.497,E2 -11870.497} C_VEL
LIN {X 0,Y 383.249,Z 333.057,A -85,B 0,C 180,E1 -11872.624,E2 -11872.624} C_VEL
LIN {X 0,Y 383.175,Z 333.063,A -85,B 0,C 180,E1 -11874.738,E2 -11874.738} C_VEL
LIN {X 0,Y 383.36,Z 333.044,A -85,B 0,C 180,E1 -11877.898,E2 -11877.898} C_VEL
LIN {X 0,Y 383.493,Z 333.022,A -85,B 0,C 180,E1 -11880,E2 -11880} C_VEL
LIN {X 0,Y 383.263,Z 333.056,A -85,B 0,C 180,E1 -11883.153,E2 -11883.153} C_VEL
LIN {X 0,Y 383.273,Z 333.054,A -85,B 0,C 180,E1 -11886.316,E2 -11886.316} C_VEL
LIN {X 0,Y 383.236,Z 333.059,A -85,B 0,C 180,E1 -11888.436,E2 -11888.436} C_VEL
LIN {X 0,Y 383.085,Z 333.08,A -85,B 0,C 180,E1 -11891.642,E2 -11891.642} C_VEL
LIN {X 0,Y 383.09,Z 333.079,A -85,B 0,C 180,E1 -11894.882,E2 -11894.882} C_VEL
LIN {X 0,Y 383.072,Z 333.081,A -85,B 0,C 180,E1 -11898.173,E2 -11898.173} C_VEL
LIN {X 0,Y 383.052,Z 333.084,A -85,B 0,C 180,E1 -11901.527,E2 -11901.527} C_VEL
LIN {X 0,Y 383.032,Z 333.085,A -85,B 0,C 180,E1 -11904.961,E2 -11904.961} C_VEL
LIN {X 0,Y 383.018,Z 333.089,A -85,B 0,C 180,E1 -11908.494,E2 -11908.494} C_VEL
LIN {X 0,Y 382.987,Z 333.092,A -85,B 0,C 180,E1 -11912.151,E2 -11912.151} C_VEL
LIN {X 0,Y 382.997,Z 333.091,A -85,B 0,C 180,E1 -11914.67,E2 -11914.67} C_VEL
LIN {X 0,Y 383.017,Z 333.222,A -85,B 0,C 180,E1 -11916.665,E2 -11916.665} C_VEL
LIN {X 0,Y 386.038,Z 343.536,A -85,B 0,C 180,E1 -11920.329,E2 -11920.329} C_VEL
LIN {X 0,Y 388.185,Z 350.895,A -85,B 0,C 180,E1 -11922.759,E2 -11922.759} C_VEL
LIN {X 0,Y 391.29,Z 361.093,A -85,B 0,C 180,E1 -11925.926,E2 -11925.926} C_VEL
LIN {X 0,Y 394.491,Z 372.638,A -85,B 0,C 180,E1 -11929.212,E2 -11929.212} C_VEL
LIN {X 0,Y 396.507,Z 380.278,A -85,B 0,C 180,E1 -11931.25,E2 -11931.25} C_VEL
LIN {X 0,Y 395.64,Z 386.087,A -85,B 0,C 180,E1 -11932.53,E2 -11932.53} C_VEL
LIN {X 0,Y 392.689,Z 403.87,A -85,B 0,C 180,E1 -11936.306,E2 -11936.306} C_VEL
LIN {X 0,Y 390.863,Z 416.754,A -85,B 0,C 180,E1 -11938.938,E2 -11938.938} C_VEL
LIN {X 0,Y 395.303,Z 441.11,A -85,B 0,C 180,E1 -11939.88,E2 -11939.88} C_VEL
LIN {X 0,Y 397.441,Z 453.959,A -85,B 0,C 180,E1 -11940.497,E2 -11940.497} C_VEL
LIN {X 0,Y 398.079,Z 459.112,A -85,B 0,C 180,E1 -11940.772,E2 -11940.772} C_VEL
LIN {X 0,Y 396.768,Z 474.37,A -85,B 0,C 180,E1 -11941.504,E2 -11941.504} C_VEL
LIN {X 0,Y 395.107,Z 489.981,A -85,B 0,C 180,E1 -11942.456,E2 -11942.456} C_VEL
LIN {X 0,Y 393.42,Z 505.159,A -85,B 0,C 180,E1 -11943.621,E2 -11943.621} C_VEL
LIN {X 0,Y 391.552,Z 519.167,A -85,B 0,C 180,E1 -11944.913,E2 -11944.913} C_VEL
LIN {X 0,Y 389.638,Z 533.353,A -85,B 0,C 180,E1 -11946.483,E2 -11946.483} C_VEL
LIN {X 0,Y 387.848,Z 546.33,A -85,B 0,C 180,E1 -11948.197,E2 -11948.197} C_VEL
LIN {X 0,Y 386.251,Z 558.207,A -85,B 0,C 180,E1 -11950.055,E2 -11950.055} C_VEL
LIN {X 0,Y 384.913,Z 568.338,A -85,B 0,C 180,E1 -11951.92,E2 -11951.92} C_VEL
LIN {X 0,Y 383.995,Z 576.938,A -85,B 0,C 180,E1 -11953.796,E2 -11953.796} C_VEL
LIN {X 0,Y 383.131,Z 584.322,A -85,B 0,C 180,E1 -11955.665,E2 -11955.665} C_VEL
LIN {X 0,Y 382.549,Z 591.399,A -85,B 0,C 180,E1 -11957.806,E2 -11957.806} C_VEL
LIN {X 0,Y 382.131,Z 597.111,A -85,B 0,C 180,E1 -11959.94,E2 -11959.94} C_VEL
LIN {X 0,Y 382.017,Z 600.646,A -85,B 0,C 180,E1 -11961.539,E2 -11961.539} C_VEL
LIN {X 0,Y 381.971,Z 604.325,A -85,B 0,C 180,E1 -11963.665,E2 -11963.665} C_VEL
LIN {X 0,Y 381.9,Z 606.915,A -85,B 0,C 180,E1 -11965.781,E2 -11965.781} C_VEL
LIN {X 0,Y 381.927,Z 608.382,A -85,B 0,C 180,E1 -11967.893,E2 -11967.893} C_VEL
LIN {X 0,Y 381.895,Z 608.858,A -85,B 0,C 180,E1 -11970.003,E2 -11970.003} C_VEL
LIN {X 0,Y 381.946,Z 608.202,A -85,B 0,C 180,E1 -11972.112,E2 -11972.112} C_VEL
LIN {X 0,Y 381.918,Z 606.555,A -85,B 0,C 180,E1 -11974.224,E2 -11974.224} C_VEL
LIN {X 0,Y 382.036,Z 603.37,A -85,B 0,C 180,E1 -11976.594,E2 -11976.594} C_VEL
LIN {X 0,Y 382.095,Z 599.876,A -85,B 0,C 180,E1 -11978.464,E2 -11978.464} C_VEL
LIN {X 0,Y 382.26,Z 594.784,A -85,B 0,C 180,E1 -11980.597,E2 -11980.597} C_VEL
LIN {X 0,Y 382.765,Z 588.437,A -85,B 0,C 180,E1 -11982.731,E2 -11982.731} C_VEL
LIN {X 0,Y 383.369,Z 580.724,A -85,B 0,C 180,E1 -11984.874,E2 -11984.874} C_VEL
LIN {X 0,Y 384.381,Z 571.514,A -85,B 0,C 180,E1 -11987.013,E2 -11987.013} C_VEL
LIN {X 0,Y 385.622,Z 560.473,A -85,B 0,C 180,E1 -11989.153,E2 -11989.153} C_VEL
LIN {X 0,Y 387.04,Z 549.078,A -85,B 0,C 180,E1 -11991.018,E2 -11991.018} C_VEL
LIN {X 0,Y 388.711,Z 536.539,A -85,B 0,C 180,E1 -11992.767,E2 -11992.767} C_VEL
LIN {X 0,Y 390.574,Z 522.304,A -85,B 0,C 180,E1 -11994.45,E2 -11994.45} C_VEL
LIN {X 0,Y 392.479,Z 507.863,A -85,B 0,C 180,E1 -11995.881,E2 -11995.881} C_VEL
LIN {X 0,Y 394.314,Z 492.793,A -85,B 0,C 180,E1 -11997.13,E2 -11997.13} C_VEL
LIN {X 0,Y 396.015,Z 478.263,A -85,B 0,C 180,E1 -11998.127,E2 -11998.127} C_VEL
LIN {X 0,Y 397.423,Z 463.722,A -85,B 0,C 180,E1 -11998.937,E2 -11998.937} C_VEL
LIN {X 0,Y 397.859,Z 457.784,A -85,B 0,C 180,E1 -11999.228,E2 -11999.228} C_VEL
LIN {X 0,Y 395.667,Z 442.189,A -85,B 0,C 180,E1 -12000.135,E2 -12000.135} C_VEL
LIN {X 0,Y 393.899,Z 428.343,A -85,B 0,C 180,E1 -12000.786,E2 -12000.786} C_VEL
LIN {X 0,Y 391.011,Z 413.653,A -85,B 0,C 180,E1 -12001.53,E2 -12001.53} C_VEL
LIN {X 0,Y 393.68,Z 399.061,A -85,B 0,C 180,E1 -12004.841,E2 -12004.841} C_VEL
LIN {X 0,Y 396.896,Z 386.691,A -85,B 0,C 180,E1 -12007.978,E2 -12007.978} C_VEL
LIN {X 0,Y 397.764,Z 383.229,A -85,B 0,C 180,E1 -12008.975,E2 -12008.975} C_VEL
LIN {X 0,Y 396.638,Z 378.3,A -85,B 0,C 180,E1 -12010.967,E2 -12010.967} C_VEL
LIN {X 0,Y 395.339,Z 373.971,A -85,B 0,C 180,E1 -12013.209,E2 -12013.209} C_VEL
LIN {X 0,Y 394.169,Z 370.723,A -85,B 0,C 180,E1 -12015.498,E2 -12015.498} C_VEL
LIN {X 0,Y 393.462,Z 369.005,A -85,B 0,C 180,E1 -12017.254,E2 -12017.254} C_VEL
LIN {X 0,Y 392.568,Z 367.635,A -85,B 0,C 180,E1 -12019.873,E2 -12019.873} C_VEL
LIN {X 0,Y 391.823,Z 367.509,A -85,B 0,C 180,E1 -12022.422,E2 -12022.422} C_VEL
LIN {X 0,Y 390.75,Z 368.57,A -85,B 0,C 180,E1 -12024.862,E2 -12024.862} C_VEL
LIN {X 0,Y 389.218,Z 371.096,A -85,B 0,C 180,E1 -12028.07,E2 -12028.07} C_VEL
LIN {X 0,Y 388.269,Z 373.77,A -85,B 0,C 180,E1 -12030.744,E2 -12030.744} C_VEL
LIN {X 0,Y 387.267,Z 377.803,A -85,B 0,C 180,E1 -12034.181,E2 -12034.181} C_VEL
LIN {X 0,Y 386.55,Z 382.248,A -85,B 0,C 180,E1 -12037.555,E2 -12037.555} C_VEL
LIN {X 0,Y 392.374,Z 395.77,A -85,B 0,C 180,E1 -12039.114,E2 -12039.114} C_VEL
LIN {X 0,Y 395.829,Z 406.567,A -85,B 0,C 180,E1 -12040.285,E2 -12040.285} C_VEL
LIN {X 0,Y 394.245,Z 421.109,A -85,B 0,C 180,E1 -12041.419,E2 -12041.419} C_VEL
LIN {X 0,Y 392.815,Z 433.072,A -85,B 0,C 180,E1 -12042.562,E2 -12042.562} C_VEL
LIN {X 0,Y 391.268,Z 445.049,A -85,B 0,C 180,E1 -12043.969,E2 -12043.969} C_VEL
LIN {X 0,Y 389.941,Z 455.061,A -85,B 0,C 180,E1 -12045.385,E2 -12045.385} C_VEL
LIN {X 0,Y 388.704,Z 464.033,A -85,B 0,C 180,E1 -12046.938,E2 -12046.938} C_VEL
LIN {X 0,Y 387.565,Z 471.467,A -85,B 0,C 180,E1 -12048.494,E2 -12048.494} C_VEL
LIN {X 0,Y 386.601,Z 477.529,A -85,B 0,C 180,E1 -12050.056,E2 -12050.056} C_VEL
LIN {X 0,Y 385.697,Z 482.395,A -85,B 0,C 180,E1 -12051.618,E2 -12051.618} C_VEL
LIN {X 0,Y 385.102,Z 486.167,A -85,B 0,C 180,E1 -12053.188,E2 -12053.188} C_VEL
LIN {X 0,Y 384.73,Z 488.9,A -85,B 0,C 180,E1 -12054.76,E2 -12054.76} C_VEL
LIN {X 0,Y 384.408,Z 490.188,A -85,B 0,C 180,E1 -12055.807,E2 -12055.807} C_VEL
LIN {X 0,Y 384.159,Z 491.064,A -85,B 0,C 180,E1 -12056.854,E2 -12056.854} C_VEL
LIN {X 0,Y 383.875,Z 491.563,A -85,B 0,C 180,E1 -12057.902,E2 -12057.902} C_VEL
LIN {X 0,Y 383.724,Z 491.646,A -85,B 0,C 180,E1 -12058.951,E2 -12058.951} C_VEL
LIN {X 0,Y 383.564,Z 491.297,A -85,B 0,C 180,E1 -12060,E2 -12060} C_VEL
LIN {X 0,Y 383.504,Z 490.524,A -85,B 0,C 180,E1 -12061.05,E2 -12061.05} C_VEL
LIN {X 0,Y 383.437,Z 489.354,A -85,B 0,C 180,E1 -12062.101,E2 -12062.101} C_VEL
LIN {X 0,Y 383.516,Z 486.784,A -85,B 0,C 180,E1 -12063.678,E2 -12063.678} C_VEL
LIN {X 0,Y 383.462,Z 483.263,A -85,B 0,C 180,E1 -12065.258,E2 -12065.258} C_VEL
LIN {X 0,Y 383.92,Z 477.731,A -85,B 0,C 180,E1 -12067.109,E2 -12067.109} C_VEL
LIN {X 0,Y 384.28,Z 471.741,A -85,B 0,C 180,E1 -12068.699,E2 -12068.699} C_VEL
LIN {X 0,Y 384.713,Z 464.55,A -85,B 0,C 180,E1 -12070.26,E2 -12070.26} C_VEL
LIN {X 0,Y 385.312,Z 455.68,A -85,B 0,C 180,E1 -12071.841,E2 -12071.841} C_VEL
LIN {X 0,Y 385.868,Z 446.828,A -85,B 0,C 180,E1 -12073.16,E2 -12073.16} C_VEL
LIN {X 0,Y 386.692,Z 436.265,A -85,B 0,C 180,E1 -12074.472,E2 -12074.472} C_VEL
LIN {X 0,Y 387.456,Z 423.424,A -85,B 0,C 180,E1 -12075.789,E2 -12075.789} C_VEL
LIN {X 0,Y 388.297,Z 410.661,A -85,B 0,C 180,E1 -12076.834,E2 -12076.834} C_VEL
LIN {X 0,Y 389.015,Z 396.657,A -85,B 0,C 180,E1 -12077.751,E2 -12077.751} C_VEL
LIN {X 0,Y 388.7,Z 393.152,A -85,B 0,C 180,E1 -12077.963,E2 -12077.963} C_VEL
LIN {X 0,Y 385.233,Z 378.663,A -85,B 0,C 180,E1 -12078.821,E2 -12078.821} C_VEL
LIN {X 0,Y 382.88,Z 369.299,A -85,B 0,C 180,E1 -12079.294,E2 -12079.294} C_VEL
LIN {X 0,Y 383.057,Z 363.133,A -85,B 0,C 180,E1 -12082.662,E2 -12082.662} C_VEL
LIN {X 0,Y 383.285,Z 356.947,A -85,B 0,C 180,E1 -12086.109,E2 -12086.109} C_VEL
LIN {X 0,Y 383.544,Z 351.737,A -85,B 0,C 180,E1 -12089.051,E2 -12089.051} C_VEL
LIN {X 0,Y 383.84,Z 345.585,A -85,B 0,C 180,E1 -12092.619,E2 -12092.619} C_VEL
LIN {X 0,Y 383.978,Z 340.107,A -85,B 0,C 180,E1 -12095.853,E2 -12095.853} C_VEL
LIN {X 0,Y 383.495,Z 335.772,A -85,B 0,C 180,E1 -12098.543,E2 -12098.543} C_VEL
LIN {X 0,Y 383.015,Z 333.092,A -85,B 0,C 180,E1 -12100.302,E2 -12100.302} C_VEL
LIN {X 0,Y 383.015,Z 333.086,A -85,B 0,C 180,E1 -12102.778,E2 -12102.778} C_VEL
LIN {X 0,Y 383.006,Z 333.091,A -85,B 0,C 180,E1 -12105.788,E2 -12105.788} C_VEL
LIN {X 0,Y 383.025,Z 333.107,A -85,B 0,C 180,E1 -12109.179,E2 -12109.179} C_VEL
LIN {X 0,Y 384.175,Z 339.105,A -85,B 0,C 180,E1 -12111.872,E2 -12111.872} C_VEL
LIN {X 0,Y 385.001,Z 344.351,A -85,B 0,C 180,E1 -12114.255,E2 -12114.255} C_VEL
LIN {X 0,Y 384.978,Z 349.875,A -85,B 0,C 180,E1 -12116.791,E2 -12116.791} C_VEL
LIN {X 0,Y 384.784,Z 357.712,A -85,B 0,C 180,E1 -12120.45,E2 -12120.45} C_VEL
LIN {X 0,Y 384.695,Z 365.359,A -85,B 0,C 180,E1 -12123.992,E2 -12123.992} C_VEL
LIN {X 0,Y 384.79,Z 373.136,A -85,B 0,C 180,E1 -12127.444,E2 -12127.444} C_VEL
LIN {X 0,Y 385.008,Z 382.446,A -85,B 0,C 180,E1 -12131.193,E2 -12131.193} C_VEL
LIN {X 0,Y 385.11,Z 383.064,A -85,B 0,C 180,E1 -12131.28,E2 -12131.28} C_VEL
LIN {X 0,Y 388.943,Z 395.165,A -85,B 0,C 180,E1 -12131.848,E2 -12131.848} C_VEL
LIN {X 0,Y 389.806,Z 398.941,A -85,B 0,C 180,E1 -12132.048,E2 -12132.048} C_VEL
LIN {X 0,Y 389.412,Z 411.2,A -85,B 0,C 180,E1 -12132.673,E2 -12132.673} C_VEL
LIN {X 0,Y 388.883,Z 423.793,A -85,B 0,C 180,E1 -12133.555,E2 -12133.555} C_VEL
LIN {X 0,Y 388.178,Z 434.403,A -85,B 0,C 180,E1 -12134.509,E2 -12134.509} C_VEL
LIN {X 0,Y 387.421,Z 444.759,A -85,B 0,C 180,E1 -12135.688,E2 -12135.688} C_VEL
LIN {X 0,Y 386.587,Z 454.931,A -85,B 0,C 180,E1 -12137.13,E2 -12137.13} C_VEL
LIN {X 0,Y 385.701,Z 463.743,A -85,B 0,C 180,E1 -12138.702,E2 -12138.702} C_VEL
LIN {X 0,Y 385.135,Z 470.461,A -85,B 0,C 180,E1 -12140.2,E2 -12140.2} C_VEL
LIN {X 0,Y 384.654,Z 475.554,A -85,B 0,C 180,E1 -12141.593,E2 -12141.593} C_VEL
LIN {X 0,Y 383.897,Z 480.216,A -85,B 0,C 180,E1 -12143.163,E2 -12143.163} C_VEL
LIN {X 0,Y 383.594,Z 483.737,A -85,B 0,C 180,E1 -12144.741,E2 -12144.741} C_VEL
LIN {X 0,Y 383.535,Z 485.535,A -85,B 0,C 180,E1 -12145.794,E2 -12145.794} C_VEL
LIN {X 0,Y 383.45,Z 486.914,A -85,B 0,C 180,E1 -12146.846,E2 -12146.846} C_VEL
LIN {X 0,Y 383.164,Z 488.506,A -85,B 0,C 180,E1 -12148.946,E2 -12148.946} C_VEL
LIN {X 0,Y 383.126,Z 488.739,A -85,B 0,C 180,E1 -12149.997,E2 -12149.997} C_VEL
LIN {X 0,Y 383.273,Z 487.972,A -85,B 0,C 180,E1 -12152.099,E2 -12152.099} C_VEL
LIN {X 0,Y 383.46,Z 487.016,A -85,B 0,C 180,E1 -12153.149,E2 -12153.149} C_VEL
LIN {X 0,Y 383.548,Z 485.694,A -85,B 0,C 180,E1 -12154.201,E2 -12154.201} C_VEL
LIN {X 0,Y 383.75,Z 482.907,A -85,B 0,C 180,E1 -12155.778,E2 -12155.778} C_VEL
LIN {X 0,Y 384.18,Z 479.093,A -85,B 0,C 180,E1 -12157.354,E2 -12157.354} C_VEL
LIN {X 0,Y 384.799,Z 474.136,A -85,B 0,C 180,E1 -12158.928,E2 -12158.928} C_VEL
LIN {X 0,Y 385.33,Z 467.911,A -85,B 0,C 180,E1 -12160.506,E2 -12160.506} C_VEL
LIN {X 0,Y 386.111,Z 460.141,A -85,B 0,C 180,E1 -12162.08,E2 -12162.08} C_VEL
LIN {X 0,Y 386.909,Z 452.18,A -85,B 0,C 180,E1 -12163.388,E2 -12163.388} C_VEL
LIN {X 0,Y 387.575,Z 443.508,A -85,B 0,C 180,E1 -12164.569,E2 -12164.569} C_VEL
LIN {X 0,Y 387.957,Z 438.338,A -85,B 0,C 180,E1 -12165.169,E2 -12165.169} C_VEL
LIN {X 0,Y 387.642,Z 433.643,A -85,B 0,C 180,E1 -12165.698,E2 -12165.698} C_VEL
LIN {X 0,Y 385.45,Z 425.898,A -85,B 0,C 180,E1 -12166.564,E2 -12166.564} C_VEL
LIN {X 0,Y 383.163,Z 417.81,A -85,B 0,C 180,E1 -12167.339,E2 -12167.339} C_VEL
LIN {X 0,Y 382.751,Z 412.529,A -85,B 0,C 180,E1 -12167.72,E2 -12167.72} C_VEL
LIN {X 0,Y 383.15,Z 400.419,A -85,B 0,C 180,E1 -12168.356,E2 -12168.356} C_VEL
LIN {X 0,Y 381.701,Z 394.529,A -85,B 0,C 180,E1 -12168.676,E2 -12168.676} C_VEL
LIN {X 0,Y 378.107,Z 383.577,A -85,B 0,C 180,E1 -12169.228,E2 -12169.228} C_VEL
LIN {X 0,Y 377.941,Z 375.604,A -85,B 0,C 180,E1 -12172.405,E2 -12172.405} C_VEL
LIN {X 0,Y 377.824,Z 367.607,A -85,B 0,C 180,E1 -12175.917,E2 -12175.917} C_VEL
LIN {X 0,Y 377.937,Z 359.798,A -85,B 0,C 180,E1 -12179.52,E2 -12179.52} C_VEL
LIN {X 0,Y 378.049,Z 353.209,A -85,B 0,C 180,E1 -12182.62,E2 -12182.62} C_VEL
LIN {X 0,Y 378.159,Z 347.634,A -85,B 0,C 180,E1 -12185.175,E2 -12185.175} C_VEL
LIN {X 0,Y 377.695,Z 343.013,A -85,B 0,C 180,E1 -12187.321,E2 -12187.321} C_VEL
LIN {X 0,Y 376.545,Z 336.992,A -85,B 0,C 180,E1 -12190.071,E2 -12190.071} C_VEL
LIN {X 0,Y 375.94,Z 333.972,A -85,B 0,C 180,E1 -12191.458,E2 -12191.458} C_VEL
LIN {X 0,Y 375.964,Z 333.969,A -85,B 0,C 180,E1 -12195.258,E2 -12195.258} C_VEL
LIN {X 0,Y 375.975,Z 333.965,A -85,B 0,C 180,E1 -12198.387,E2 -12198.387} C_VEL
LIN {X 0,Y 375.952,Z 333.966,A -85,B 0,C 180,E1 -12201.909,E2 -12201.909} C_VEL
LIN {X 0,Y 375.962,Z 333.967,A -85,B 0,C 180,E1 -12205.33,E2 -12205.33} C_VEL
LIN {X 0,Y 375.938,Z 333.97,A -85,B 0,C 180,E1 -12208.436,E2 -12208.436} C_VEL
LIN {X 0,Y 375.963,Z 333.967,A -85,B 0,C 180,E1 -12212.138,E2 -12212.138} C_VEL
LIN {X 0,Y 375.988,Z 333.962,A -85,B 0,C 180,E1 -12214.537,E2 -12214.537} C_VEL
LIN {X 0,Y 376.004,Z 333.958,A -85,B 0,C 180,E1 -12218.048,E2 -12218.048} C_VEL
LIN {X 0,Y 376.009,Z 333.953,A -85,B 0,C 180,E1 -12221.473,E2 -12221.473} C_VEL
LIN {X 0,Y 376.037,Z 333.951,A -85,B 0,C 180,E1 -12224.831,E2 -12224.831} C_VEL
LIN {X 0,Y 376.041,Z 333.958,A -85,B 0,C 180,E1 -12228.136,E2 -12228.136} C_VEL
LIN {X 0,Y 376.234,Z 333.929,A -85,B 0,C 180,E1 -12231.876,E2 -12231.876} C_VEL
LIN {X 0,Y 376.147,Z 333.938,A -85,B 0,C 180,E1 -12234.639,E2 -12234.639} C_VEL
LIN {X 0,Y 376.326,Z 333.92,A -85,B 0,C 180,E1 -12237.859,E2 -12237.859} C_VEL
LIN {X 0,Y 376.463,Z 333.898,A -85,B 0,C 180,E1 -12240,E2 -12240} C_VEL
LIN {X 0,Y 376.199,Z 333.936,A -85,B 0,C 180,E1 -12243.212,E2 -12243.212} C_VEL
LIN {X 0,Y 376.23,Z 333.931,A -85,B 0,C 180,E1 -12246.435,E2 -12246.435} C_VEL
LIN {X 0,Y 376.182,Z 333.938,A -85,B 0,C 180,E1 -12248.595,E2 -12248.595} C_VEL
LIN {X 0,Y 376.036,Z 333.957,A -85,B 0,C 180,E1 -12251.863,E2 -12251.863} C_VEL
LIN {X 0,Y 376.038,Z 333.957,A -85,B 0,C 180,E1 -12255.168,E2 -12255.168} C_VEL
LIN {X 0,Y 376.009,Z 333.96,A -85,B 0,C 180,E1 -12258.526,E2 -12258.526} C_VEL
LIN {X 0,Y 376.002,Z 333.961,A -85,B 0,C 180,E1 -12261.951,E2 -12261.951} C_VEL
LIN {X 0,Y 375.985,Z 333.964,A -85,B 0,C 180,E1 -12265.462,E2 -12265.462} C_VEL
LIN {X 0,Y 375.948,Z 333.967,A -85,B 0,C 180,E1 -12269.081,E2 -12269.081} C_VEL
LIN {X 0,Y 375.928,Z 333.971,A -85,B 0,C 180,E1 -12272.83,E2 -12272.83} C_VEL
LIN {X 0,Y 375.988,Z 334.128,A -85,B 0,C 180,E1 -12275.818,E2 -12275.818} C_VEL
LIN {X 0,Y 379.123,Z 344.921,A -85,B 0,C 180,E1 -12279.757,E2 -12279.757} C_VEL
LIN {X 0,Y 381.85,Z 354.334,A -85,B 0,C 180,E1 -12282.921,E2 -12282.921} C_VEL
LIN {X 0,Y 384.913,Z 364.394,A -85,B 0,C 180,E1 -12286.071,E2 -12286.071} C_VEL
LIN {X 0,Y 388.161,Z 376.355,A -85,B 0,C 180,E1 -12289.503,E2 -12289.503} C_VEL
LIN {X 0,Y 389.728,Z 382.249,A -85,B 0,C 180,E1 -12291.097,E2 -12291.097} C_VEL
LIN {X 0,Y 388.73,Z 388.502,A -85,B 0,C 180,E1 -12292.497,E2 -12292.497} C_VEL
LIN {X 0,Y 385.52,Z 407.171,A -85,B 0,C 180,E1 -12296.537,E2 -12296.537} C_VEL
LIN {X 0,Y 384.161,Z 416.152,A -85,B 0,C 180,E1 -12298.428,E2 -12298.428} C_VEL
LIN {X 0,Y 388.658,Z 441.483,A -85,B 0,C 180,E1 -12299.453,E2 -12299.453} C_VEL
LIN {X 0,Y 391.011,Z 456.053,A -85,B 0,C 180,E1 -12300.187,E2 -12300.187} C_VEL
LIN {X 0,Y 391.429,Z 460.226,A -85,B 0,C 180,E1 -12300.416,E2 -12300.416} C_VEL
LIN {X 0,Y 389.953,Z 476.662,A -85,B 0,C 180,E1 -12301.254,E2 -12301.254} C_VEL
LIN {X 0,Y 388.261,Z 491.588,A -85,B 0,C 180,E1 -12302.215,E2 -12302.215} C_VEL
LIN {X 0,Y 386.53,Z 506.524,A -85,B 0,C 180,E1 -12303.405,E2 -12303.405} C_VEL
LIN {X 0,Y 384.46,Z 521.525,A -85,B 0,C 180,E1 -12304.852,E2 -12304.852} C_VEL
LIN {X 0,Y 382.576,Z 534.819,A -85,B 0,C 180,E1 -12306.4,E2 -12306.4} C_VEL
LIN {X 0,Y 380.837,Z 546.853,A -85,B 0,C 180,E1 -12308.06,E2 -12308.06} C_VEL
LIN {X 0,Y 379.187,Z 558.505,A -85,B 0,C 180,E1 -12309.95,E2 -12309.95} C_VEL
LIN {X 0,Y 377.844,Z 568.466,A -85,B 0,C 180,E1 -12311.85,E2 -12311.85} C_VEL
LIN {X 0,Y 376.882,Z 576.974,A -85,B 0,C 180,E1 -12313.76,E2 -12313.76} C_VEL
LIN {X 0,Y 375.959,Z 585.141,A -85,B 0,C 180,E1 -12315.938,E2 -12315.938} C_VEL
LIN {X 0,Y 375.419,Z 591.917,A -85,B 0,C 180,E1 -12318.119,E2 -12318.119} C_VEL
LIN {X 0,Y 375.018,Z 597.392,A -85,B 0,C 180,E1 -12320.293,E2 -12320.293} C_VEL
LIN {X 0,Y 374.92,Z 601.629,A -85,B 0,C 180,E1 -12322.463,E2 -12322.463} C_VEL
LIN {X 0,Y 374.829,Z 604.785,A -85,B 0,C 180,E1 -12324.623,E2 -12324.623} C_VEL
LIN {X 0,Y 374.954,Z 606.805,A -85,B 0,C 180,E1 -12326.779,E2 -12326.779} C_VEL
LIN {X 0,Y 374.871,Z 607.768,A -85,B 0,C 180,E1 -12328.928,E2 -12328.928} C_VEL
LIN {X 0,Y 374.885,Z 607.662,A -85,B 0,C 180,E1 -12331.077,E2 -12331.077} C_VEL
LIN {X 0,Y 374.958,Z 606.505,A -85,B 0,C 180,E1 -12333.226,E2 -12333.226} C_VEL
LIN {X 0,Y 374.905,Z 604.265,A -85,B 0,C 180,E1 -12335.381,E2 -12335.381} C_VEL
LIN {X 0,Y 375.014,Z 600.899,A -85,B 0,C 180,E1 -12337.541,E2 -12337.541} C_VEL
LIN {X 0,Y 375.104,Z 596.423,A -85,B 0,C 180,E1 -12339.71,E2 -12339.71} C_VEL
LIN {X 0,Y 375.591,Z 589.059,A -85,B 0,C 180,E1 -12342.429,E2 -12342.429} C_VEL
LIN {X 0,Y 376.289,Z 580.653,A -85,B 0,C 180,E1 -12344.883,E2 -12344.883} C_VEL
LIN {X 0,Y 377.297,Z 571.557,A -85,B 0,C 180,E1 -12347.063,E2 -12347.063} C_VEL
LIN {X 0,Y 378.362,Z 562.178,A -85,B 0,C 180,E1 -12348.971,E2 -12348.971} C_VEL
LIN {X 0,Y 379.79,Z 551.319,A -85,B 0,C 180,E1 -12350.871,E2 -12350.871} C_VEL
LIN {X 0,Y 381.295,Z 540.561,A -85,B 0,C 180,E1 -12352.489,E2 -12352.489} C_VEL
LIN {X 0,Y 383.19,Z 527.026,A -85,B 0,C 180,E1 -12354.231,E2 -12354.231} C_VEL
LIN {X 0,Y 385.19,Z 512.3,A -85,B 0,C 180,E1 -12355.826,E2 -12355.826} C_VEL
LIN {X 0,Y 387.149,Z 497.923,A -85,B 0,C 180,E1 -12357.126,E2 -12357.126} C_VEL
LIN {X 0,Y 389.059,Z 482.236,A -85,B 0,C 180,E1 -12358.308,E2 -12358.308} C_VEL
LIN {X 0,Y 390.839,Z 466.288,A -85,B 0,C 180,E1 -12359.278,E2 -12359.278} C_VEL
LIN {X 0,Y 391.55,Z 459.979,A -85,B 0,C 180,E1 -12359.604,E2 -12359.604} C_VEL
LIN {X 0,Y 389.529,Z 443.83,A -85,B 0,C 180,E1 -12360.595,E2 -12360.595} C_VEL
LIN {X 0,Y 387.77,Z 428.849,A -85,B 0,C 180,E1 -12361.353,E2 -12361.353} C_VEL
LIN {X 0,Y 384.554,Z 412.976,A -85,B 0,C 180,E1 -12362.227,E2 -12362.227} C_VEL
LIN {X 0,Y 387.433,Z 399.216,A -85,B 0,C 180,E1 -12365.486,E2 -12365.486} C_VEL
LIN {X 0,Y 390.863,Z 387.252,A -85,B 0,C 180,E1 -12368.672,E2 -12368.672} C_VEL
LIN {X 0,Y 391.145,Z 386.254,A -85,B 0,C 180,E1 -12368.969,E2 -12368.969} C_VEL
LIN {X 0,Y 390.58,Z 382.657,A -85,B 0,C 180,E1 -12370.376,E2 -12370.376} C_VEL
LIN {X 0,Y 389.465,Z 378.678,A -85,B 0,C 180,E1 -12372.281,E2 -12372.281} C_VEL
LIN {X 0,Y 388.035,Z 374.501,A -85,B 0,C 180,E1 -12374.942,E2 -12374.942} C_VEL
LIN {X 0,Y 387.316,Z 372.718,A -85,B 0,C 180,E1 -12376.539,E2 -12376.539} C_VEL
LIN {X 0,Y 386.393,Z 370.936,A -85,B 0,C 180,E1 -12379.096,E2 -12379.096} C_VEL
LIN {X 0,Y 385.542,Z 370.374,A -85,B 0,C 180,E1 -12381.7,E2 -12381.7} C_VEL
LIN {X 0,Y 384.87,Z 370.729,A -85,B 0,C 180,E1 -12383.465,E2 -12383.465} C_VEL
LIN {X 0,Y 383.874,Z 371.746,A -85,B 0,C 180,E1 -12385.476,E2 -12385.476} C_VEL
LIN {X 0,Y 382.201,Z 374.579,A -85,B 0,C 180,E1 -12389.012,E2 -12389.012} C_VEL
LIN {X 0,Y 380.992,Z 378.235,A -85,B 0,C 180,E1 -12392.538,E2 -12392.538} C_VEL
LIN {X 0,Y 380.123,Z 382.411,A -85,B 0,C 180,E1 -12395.999,E2 -12395.999} C_VEL
LIN {X 0,Y 379.966,Z 383.388,A -85,B 0,C 180,E1 -12396.755,E2 -12396.755} C_VEL
LIN {X 0,Y 381.328,Z 386.559,A -85,B 0,C 180,E1 -12397.152,E2 -12397.152} C_VEL
LIN {X 0,Y 385.624,Z 396.178,A -85,B 0,C 180,E1 -12398.357,E2 -12398.357} C_VEL
LIN {X 0,Y 389.081,Z 406.421,A -85,B 0,C 180,E1 -12399.548,E2 -12399.548} C_VEL
LIN {X 0,Y 389.778,Z 409.189,A -85,B 0,C 180,E1 -12399.861,E2 -12399.861} C_VEL
LIN {X 0,Y 388.098,Z 423.071,A -85,B 0,C 180,E1 -12400.977,E2 -12400.977} C_VEL
LIN {X 0,Y 386.387,Z 435.87,A -85,B 0,C 180,E1 -12402.262,E2 -12402.262} C_VEL
LIN {X 0,Y 384.931,Z 446.596,A -85,B 0,C 180,E1 -12403.561,E2 -12403.561} C_VEL
LIN {X 0,Y 383.386,Z 457.261,A -85,B 0,C 180,E1 -12405.13,E2 -12405.13} C_VEL
LIN {X 0,Y 382.072,Z 466.052,A -85,B 0,C 180,E1 -12406.707,E2 -12406.707} C_VEL
LIN {X 0,Y 380.856,Z 473.312,A -85,B 0,C 180,E1 -12408.289,E2 -12408.289} C_VEL
LIN {X 0,Y 379.815,Z 479.256,A -85,B 0,C 180,E1 -12409.876,E2 -12409.876} C_VEL
LIN {X 0,Y 378.866,Z 484.038,A -85,B 0,C 180,E1 -12411.466,E2 -12411.466} C_VEL
LIN {X 0,Y 378.217,Z 487.692,A -85,B 0,C 180,E1 -12413.063,E2 -12413.063} C_VEL
LIN {X 0,Y 377.824,Z 490.339,A -85,B 0,C 180,E1 -12414.664,E2 -12414.664} C_VEL
LIN {X 0,Y 377.476,Z 491.589,A -85,B 0,C 180,E1 -12415.729,E2 -12415.729} C_VEL
LIN {X 0,Y 377.202,Z 492.427,A -85,B 0,C 180,E1 -12416.796,E2 -12416.796} C_VEL
LIN {X 0,Y 376.907,Z 492.877,A -85,B 0,C 180,E1 -12417.863,E2 -12417.863} C_VEL
LIN {X 0,Y 376.748,Z 492.899,A -85,B 0,C 180,E1 -12418.932,E2 -12418.932} C_VEL
LIN {X 0,Y 376.575,Z 492.492,A -85,B 0,C 180,E1 -12420,E2 -12420} C_VEL
LIN {X 0,Y 376.505,Z 491.671,A -85,B 0,C 180,E1 -12421.07,E2 -12421.07} C_VEL
LIN {X 0,Y 376.443,Z 490.455,A -85,B 0,C 180,E1 -12422.14,E2 -12422.14} C_VEL
LIN {X 0,Y 376.53,Z 487.811,A -85,B 0,C 180,E1 -12423.746,E2 -12423.746} C_VEL
LIN {X 0,Y 376.456,Z 484.216,A -85,B 0,C 180,E1 -12425.356,E2 -12425.356} C_VEL
LIN {X 0,Y 376.919,Z 478.805,A -85,B 0,C 180,E1 -12427.172,E2 -12427.172} C_VEL
LIN {X 0,Y 377.314,Z 472.586,A -85,B 0,C 180,E1 -12428.841,E2 -12428.841} C_VEL
LIN {X 0,Y 377.778,Z 465.228,A -85,B 0,C 180,E1 -12430.451,E2 -12430.451} C_VEL
LIN {X 0,Y 378.398,Z 456.248,A -85,B 0,C 180,E1 -12432.061,E2 -12432.061} C_VEL
LIN {X 0,Y 378.982,Z 447.298,A -85,B 0,C 180,E1 -12433.404,E2 -12433.404} C_VEL
LIN {X 0,Y 379.824,Z 436.628,A -85,B 0,C 180,E1 -12434.74,E2 -12434.74} C_VEL
LIN {X 0,Y 380.586,Z 424.42,A -85,B 0,C 180,E1 -12436.009,E2 -12436.009} C_VEL
LIN {X 0,Y 381.353,Z 412.541,A -85,B 0,C 180,E1 -12437.012,E2 -12437.012} C_VEL
LIN {X 0,Y 382.201,Z 397.761,A -85,B 0,C 180,E1 -12438.009,E2 -12438.009} C_VEL
LIN {X 0,Y 381.821,Z 394.165,A -85,B 0,C 180,E1 -12438.235,E2 -12438.235} C_VEL
LIN {X 0,Y 378.408,Z 379.695,A -85,B 0,C 180,E1 -12439.121,E2 -12439.121} C_VEL
LIN {X 0,Y 375.87,Z 369.705,A -85,B 0,C 180,E1 -12439.633,E2 -12439.633} C_VEL
LIN {X 0,Y 376.046,Z 363.407,A -85,B 0,C 180,E1 -12443.109,E2 -12443.109} C_VEL
LIN {X 0,Y 376.293,Z 357.743,A -85,B 0,C 180,E1 -12446.296,E2 -12446.296} C_VEL
LIN {X 0,Y 376.561,Z 351.883,A -85,B 0,C 180,E1 -12449.643,E2 -12449.643} C_VEL
LIN {X 0,Y 376.864,Z 346.248,A -85,B 0,C 180,E1 -12452.943,E2 -12452.943} C_VEL
LIN {X 0,Y 376.983,Z 341.212,A -85,B 0,C 180,E1 -12455.962,E2 -12455.962} C_VEL
LIN {X 0,Y 376.547,Z 337.356,A -85,B 0,C 180,E1 -12458.378,E2 -12458.378} C_VEL
LIN {X 0,Y 375.977,Z 333.967,A -85,B 0,C 180,E1 -12460.622,E2 -12460.622} C_VEL
LIN {X 0,Y 375.939,Z 333.972,A -85,B 0,C 180,E1 -12463.765,E2 -12463.765} C_VEL
LIN {X 0,Y 375.943,Z 333.968,A -85,B 0,C 180,E1 -12466.81,E2 -12466.81} C_VEL
LIN {X 0,Y 375.963,Z 334.085,A -85,B 0,C 180,E1 -12468.769,E2 -12468.769} C_VEL
LIN {X 0,Y 377.202,Z 340.103,A -85,B 0,C 180,E1 -12471.494,E2 -12471.494} C_VEL
LIN {X 0,Y 378.11,Z 345.925,A -85,B 0,C 180,E1 -12474.16,E2 -12474.16} C_VEL
LIN {X 0,Y 378.077,Z 351.559,A -85,B 0,C 180,E1 -12476.773,E2 -12476.773} C_VEL
LIN {X 0,Y 377.895,Z 359.551,A -85,B 0,C 180,E1 -12480.471,E2 -12480.471} C_VEL
LIN {X 0,Y 377.799,Z 367.34,A -85,B 0,C 180,E1 -12484.075,E2 -12484.075} C_VEL
LIN {X 0,Y 377.893,Z 373.965,A -85,B 0,C 180,E1 -12487.009,E2 -12487.009} C_VEL
LIN {X 0,Y 378.056,Z 382.435,A -85,B 0,C 180,E1 -12490.448,E2 -12490.448} C_VEL
LIN {X 0,Y 378.148,Z 383.762,A -85,B 0,C 180,E1 -12490.915,E2 -12490.915} C_VEL
LIN {X 0,Y 382.088,Z 396.051,A -85,B 0,C 180,E1 -12491.503,E2 -12491.503} C_VEL
LIN {X 0,Y 383.108,Z 400.127,A -85,B 0,C 180,E1 -12491.729,E2 -12491.729} C_VEL
LIN {X 0,Y 382.724,Z 412.255,A -85,B 0,C 180,E1 -12492.36,E2 -12492.36} C_VEL
LIN {X 0,Y 382.16,Z 424.801,A -85,B 0,C 180,E1 -12493.253,E2 -12493.253} C_VEL
LIN {X 0,Y 381.419,Z 435.471,A -85,B 0,C 180,E1 -12494.227,E2 -12494.227} C_VEL
LIN {X 0,Y 380.628,Z 445.83,A -85,B 0,C 180,E1 -12495.427,E2 -12495.427} C_VEL
LIN {X 0,Y 379.757,Z 456.003,A -85,B 0,C 180,E1 -12496.894,E2 -12496.894} C_VEL
LIN {X 0,Y 378.826,Z 464.818,A -85,B 0,C 180,E1 -12498.494,E2 -12498.494} C_VEL
LIN {X 0,Y 378.212,Z 471.534,A -85,B 0,C 180,E1 -12500.018,E2 -12500.018} C_VEL
LIN {X 0,Y 377.723,Z 476.629,A -85,B 0,C 180,E1 -12501.437,E2 -12501.437} C_VEL
LIN {X 0,Y 376.931,Z 481.293,A -85,B 0,C 180,E1 -12503.036,E2 -12503.036} C_VEL
LIN {X 0,Y 376.607,Z 484.814,A -85,B 0,C 180,E1 -12504.644,E2 -12504.644} C_VEL
LIN {X 0,Y 376.535,Z 486.612,A -85,B 0,C 180,E1 -12505.716,E2 -12505.716} C_VEL
LIN {X 0,Y 376.448,Z 487.991,A -85,B 0,C 180,E1 -12506.787,E2 -12506.787} C_VEL
LIN {X 0,Y 376.148,Z 489.583,A -85,B 0,C 180,E1 -12508.927,E2 -12508.927} C_VEL
LIN {X 0,Y 376.109,Z 489.816,A -85,B 0,C 180,E1 -12509.997,E2 -12509.997} C_VEL
LIN {X 0,Y 376.261,Z 489.048,A -85,B 0,C 180,E1 -12512.138,E2 -12512.138} C_VEL
LIN {X 0,Y 376.458,Z 488.091,A -85,B 0,C 180,E1 -12513.208,E2 -12513.208} C_VEL
LIN {X 0,Y 376.546,Z 486.77,A -85,B 0,C 180,E1 -12514.279,E2 -12514.279} C_VEL
LIN {X 0,Y 376.766,Z 483.982,A -85,B 0,C 180,E1 -12515.886,E2 -12515.886} C_VEL
LIN {X 0,Y 377.223,Z 480.167,A -85,B 0,C 180,E1 -12517.491,E2 -12517.491} C_VEL
LIN {X 0,Y 377.876,Z 475.207,A -85,B 0,C 180,E1 -12519.093,E2 -12519.093} C_VEL
LIN {X 0,Y 378.428,Z 468.983,A -85,B 0,C 180,E1 -12520.7,E2 -12520.7} C_VEL
LIN {X 0,Y 379.248,Z 461.21,A -85,B 0,C 180,E1 -12522.302,E2 -12522.302} C_VEL
LIN {X 0,Y 380.084,Z 453.247,A -85,B 0,C 180,E1 -12523.633,E2 -12523.633} C_VEL
LIN {X 0,Y 380.786,Z 444.57,A -85,B 0,C 180,E1 -12524.835,E2 -12524.835} C_VEL
LIN {X 0,Y 381.534,Z 433.807,A -85,B 0,C 180,E1 -12526.037,E2 -12526.037} C_VEL
LIN {X 0,Y 382.282,Z 422.136,A -85,B 0,C 180,E1 -12527.061,E2 -12527.061} C_VEL
LIN {X 0,Y 382.751,Z 412.529,A -85,B 0,C 180,E1 -12527.72,E2 -12527.72} C_VEL
LIN {X 0,Y 382.527,Z 408.935,A -85,B 0,C 180,E1 -12527.957,E2 -12527.957} C_VEL
LIN {X 0,Y 380.937,Z 403.791,A -85,B 0,C 180,E1 -12528.331,E2 -12528.331} C_VEL
LIN {X 0,Y 378.439,Z 398.928,A -85,B 0,C 180,E1 -12528.702,E2 -12528.702} C_VEL
LIN {X 0,Y 374.575,Z 392.383,A -85,B 0,C 180,E1 -12529.165,E2 -12529.165} C_VEL
LIN {X 0,Y 372.054,Z 387.157,A -85,B 0,C 180,E1 -12529.455,E2 -12529.455} C_VEL
LIN {X 0,Y 371.398,Z 385.304,A -85,B 0,C 180,E1 -12529.536,E2 -12529.536} C_VEL
LIN {X 0,Y 371.252,Z 384.618,A -85,B 0,C 180,E1 -12529.579,E2 -12529.579} C_VEL
LIN {X 0,Y 371.057,Z 376.472,A -85,B 0,C 180,E1 -12532.844,E2 -12532.844} C_VEL
LIN {X 0,Y 370.978,Z 368.29,A -85,B 0,C 180,E1 -12536.432,E2 -12536.432} C_VEL
LIN {X 0,Y 371.071,Z 360.349,A -85,B 0,C 180,E1 -12540.122,E2 -12540.122} C_VEL
LIN {X 0,Y 371.218,Z 352.882,A -85,B 0,C 180,E1 -12543.589,E2 -12543.589} C_VEL
LIN {X 0,Y 371.242,Z 347.86,A -85,B 0,C 180,E1 -12545.93,E2 -12545.93} C_VEL
LIN {X 0,Y 370.285,Z 341.732,A -85,B 0,C 180,E1 -12548.776,E2 -12548.776} C_VEL
LIN {X 0,Y 368.883,Z 334.849,A -85,B 0,C 180,E1 -12551.92,E2 -12551.92} C_VEL
LIN {X 0,Y 368.939,Z 334.844,A -85,B 0,C 180,E1 -12555.184,E2 -12555.184} C_VEL
LIN {X 0,Y 368.926,Z 334.842,A -85,B 0,C 180,E1 -12558.183,E2 -12558.183} C_VEL
LIN {X 0,Y 368.898,Z 334.846,A -85,B 0,C 180,E1 -12561.356,E2 -12561.356} C_VEL
LIN {X 0,Y 368.919,Z 334.843,A -85,B 0,C 180,E1 -12565.144,E2 -12565.144} C_VEL
LIN {X 0,Y 368.91,Z 334.845,A -85,B 0,C 180,E1 -12569.044,E2 -12569.044} C_VEL
LIN {X 0,Y 368.956,Z 334.839,A -85,B 0,C 180,E1 -12571.561,E2 -12571.561} C_VEL
LIN {X 0,Y 368.98,Z 334.829,A -85,B 0,C 180,E1 -12574.018,E2 -12574.018} C_VEL
LIN {X 0,Y 368.957,Z 334.831,A -85,B 0,C 180,E1 -12577.606,E2 -12577.606} C_VEL
LIN {X 0,Y 368.971,Z 334.83,A -85,B 0,C 180,E1 -12581.106,E2 -12581.106} C_VEL
LIN {X 0,Y 368.976,Z 334.835,A -85,B 0,C 180,E1 -12584.534,E2 -12584.534} C_VEL
LIN {X 0,Y 368.994,Z 334.834,A -85,B 0,C 180,E1 -12587.906,E2 -12587.906} C_VEL
LIN {X 0,Y 369.205,Z 334.803,A -85,B 0,C 180,E1 -12591.8,E2 -12591.8} C_VEL
LIN {X 0,Y 369.12,Z 334.813,A -85,B 0,C 180,E1 -12594.537,E2 -12594.537} C_VEL
LIN {X 0,Y 369.291,Z 334.797,A -85,B 0,C 180,E1 -12597.818,E2 -12597.818} C_VEL
LIN {X 0,Y 369.433,Z 334.773,A -85,B 0,C 180,E1 -12600,E2 -12600} C_VEL
LIN {X 0,Y 369.138,Z 334.815,A -85,B 0,C 180,E1 -12603.274,E2 -12603.274} C_VEL
LIN {X 0,Y 369.191,Z 334.807,A -85,B 0,C 180,E1 -12606.558,E2 -12606.558} C_VEL
LIN {X 0,Y 369.115,Z 334.819,A -85,B 0,C 180,E1 -12608.761,E2 -12608.761} C_VEL
LIN {X 0,Y 368.99,Z 334.835,A -85,B 0,C 180,E1 -12612.093,E2 -12612.093} C_VEL
LIN {X 0,Y 368.977,Z 334.836,A -85,B 0,C 180,E1 -12615.465,E2 -12615.465} C_VEL
LIN {X 0,Y 368.97,Z 334.837,A -85,B 0,C 180,E1 -12618.893,E2 -12618.893} C_VEL
LIN {X 0,Y 368.955,Z 334.838,A -85,B 0,C 180,E1 -12622.393,E2 -12622.393} C_VEL
LIN {X 0,Y 368.977,Z 334.835,A -85,B 0,C 180,E1 -12625.981,E2 -12625.981} C_VEL
LIN {X 0,Y 368.937,Z 334.841,A -85,B 0,C 180,E1 -12628.812,E2 -12628.812} C_VEL
LIN {X 0,Y 368.876,Z 334.85,A -85,B 0,C 180,E1 -12632.24,E2 -12632.24} C_VEL
LIN {X 0,Y 368.937,Z 334.917,A -85,B 0,C 180,E1 -12634.904,E2 -12634.904} C_VEL
LIN {X 0,Y 371.755,Z 344.674,A -85,B 0,C 180,E1 -12638.598,E2 -12638.598} C_VEL
LIN {X 0,Y 374.41,Z 353.793,A -85,B 0,C 180,E1 -12641.786,E2 -12641.786} C_VEL
LIN {X 0,Y 377.675,Z 364.914,A -85,B 0,C 180,E1 -12645.379,E2 -12645.379} C_VEL
LIN {X 0,Y 380.447,Z 374.768,A -85,B 0,C 180,E1 -12648.32,E2 -12648.32} C_VEL
LIN {X 0,Y 382.95,Z 384.295,A -85,B 0,C 180,E1 -12650.972,E2 -12650.972} C_VEL
LIN {X 0,Y 381.203,Z 394.111,A -85,B 0,C 180,E1 -12653.193,E2 -12653.193} C_VEL
LIN {X 0,Y 378.145,Z 411.636,A -85,B 0,C 180,E1 -12657.036,E2 -12657.036} C_VEL
LIN {X 0,Y 377.477,Z 415.876,A -85,B 0,C 180,E1 -12657.949,E2 -12657.949} C_VEL
LIN {X 0,Y 381.914,Z 441.127,A -85,B 0,C 180,E1 -12658.989,E2 -12658.989} C_VEL
LIN {X 0,Y 384.344,Z 457.139,A -85,B 0,C 180,E1 -12659.817,E2 -12659.817} C_VEL
LIN {X 0,Y 384.854,Z 460.964,A -85,B 0,C 180,E1 -12660.038,E2 -12660.038} C_VEL
LIN {X 0,Y 383.36,Z 476.633,A -85,B 0,C 180,E1 -12660.863,E2 -12660.863} C_VEL
LIN {X 0,Y 381.618,Z 491.506,A -85,B 0,C 180,E1 -12661.845,E2 -12661.845} C_VEL
LIN {X 0,Y 379.838,Z 506.24,A -85,B 0,C 180,E1 -12663.047,E2 -12663.047} C_VEL
LIN {X 0,Y 377.689,Z 521.148,A -85,B 0,C 180,E1 -12664.516,E2 -12664.516} C_VEL
LIN {X 0,Y 375.661,Z 534.95,A -85,B 0,C 180,E1 -12666.161,E2 -12666.161} C_VEL
LIN {X 0,Y 373.826,Z 547.298,A -85,B 0,C 180,E1 -12667.917,E2 -12667.917} C_VEL
LIN {X 0,Y 372.144,Z 558.762,A -85,B 0,C 180,E1 -12669.843,E2 -12669.843} C_VEL
LIN {X 0,Y 370.77,Z 568.554,A -85,B 0,C 180,E1 -12671.778,E2 -12671.778} C_VEL
LIN {X 0,Y 369.794,Z 576.977,A -85,B 0,C 180,E1 -12673.723,E2 -12673.723} C_VEL
LIN {X 0,Y 368.801,Z 585.803,A -85,B 0,C 180,E1 -12676.189,E2 -12676.189} C_VEL
LIN {X 0,Y 368.275,Z 592.332,A -85,B 0,C 180,E1 -12678.444,E2 -12678.444} C_VEL
LIN {X 0,Y 367.933,Z 597.517,A -85,B 0,C 180,E1 -12680.659,E2 -12680.659} C_VEL
LIN {X 0,Y 367.882,Z 600.621,A -85,B 0,C 180,E1 -12682.318,E2 -12682.318} C_VEL
LIN {X 0,Y 367.783,Z 603.794,A -85,B 0,C 180,E1 -12684.52,E2 -12684.52} C_VEL
LIN {X 0,Y 367.924,Z 605.819,A -85,B 0,C 180,E1 -12686.718,E2 -12686.718} C_VEL
LIN {X 0,Y 367.839,Z 606.78,A -85,B 0,C 180,E1 -12688.908,E2 -12688.908} C_VEL
LIN {X 0,Y 367.854,Z 606.665,A -85,B 0,C 180,E1 -12691.097,E2 -12691.097} C_VEL
LIN {X 0,Y 367.929,Z 605.497,A -85,B 0,C 180,E1 -12693.288,E2 -12693.288} C_VEL
LIN {X 0,Y 367.861,Z 603.235,A -85,B 0,C 180,E1 -12695.484,E2 -12695.484} C_VEL
LIN {X 0,Y 367.969,Z 599.847,A -85,B 0,C 180,E1 -12697.686,E2 -12697.686} C_VEL
LIN {X 0,Y 368.044,Z 595.346,A -85,B 0,C 180,E1 -12699.898,E2 -12699.898} C_VEL
LIN {X 0,Y 368.458,Z 589.561,A -85,B 0,C 180,E1 -12702.114,E2 -12702.114} C_VEL
LIN {X 0,Y 369.042,Z 582.501,A -85,B 0,C 180,E1 -12704.336,E2 -12704.336} C_VEL
LIN {X 0,Y 369.933,Z 574.022,A -85,B 0,C 180,E1 -12706.559,E2 -12706.559} C_VEL
LIN {X 0,Y 371.121,Z 563.908,A -85,B 0,C 180,E1 -12708.782,E2 -12708.782} C_VEL
LIN {X 0,Y 372.744,Z 551.88,A -85,B 0,C 180,E1 -12710.994,E2 -12710.994} C_VEL
LIN {X 0,Y 374.578,Z 539.456,A -85,B 0,C 180,E1 -12712.914,E2 -12712.914} C_VEL
LIN {X 0,Y 376.569,Z 525.97,A -85,B 0,C 180,E1 -12714.685,E2 -12714.685} C_VEL
LIN {X 0,Y 378.682,Z 511.332,A -85,B 0,C 180,E1 -12716.304,E2 -12716.304} C_VEL
LIN {X 0,Y 380.531,Z 498.503,A -85,B 0,C 180,E1 -12717.501,E2 -12717.501} C_VEL
LIN {X 0,Y 382.521,Z 483.49,A -85,B 0,C 180,E1 -12718.687,E2 -12718.687} C_VEL
LIN {X 0,Y 384.466,Z 467.384,A -85,B 0,C 180,E1 -12719.721,E2 -12719.721} C_VEL
LIN {X 0,Y 385.157,Z 461.257,A -85,B 0,C 180,E1 -12720.051,E2 -12720.051} C_VEL
LIN {X 0,Y 383.387,Z 444.752,A -85,B 0,C 180,E1 -12721.118,E2 -12721.118} C_VEL
LIN {X 0,Y 381.826,Z 430.177,A -85,B 0,C 180,E1 -12721.915,E2 -12721.915} C_VEL
LIN {X 0,Y 378.995,Z 415.817,A -85,B 0,C 180,E1 -12722.747,E2 -12722.747} C_VEL
LIN {X 0,Y 378.236,Z 412.225,A -85,B 0,C 180,E1 -12723.004,E2 -12723.004} C_VEL
LIN {X 0,Y 381.21,Z 399.488,A -85,B 0,C 180,E1 -12726.156,E2 -12726.156} C_VEL
LIN {X 0,Y 384.502,Z 388.913,A -85,B 0,C 180,E1 -12729.096,E2 -12729.096} C_VEL
LIN {X 0,Y 384.434,Z 386.886,A -85,B 0,C 180,E1 -12729.842,E2 -12729.842} C_VEL
LIN {X 0,Y 383.199,Z 382.194,A -85,B 0,C 180,E1 -12732.031,E2 -12732.031} C_VEL
LIN {X 0,Y 381.887,Z 378.375,A -85,B 0,C 180,E1 -12734.375,E2 -12734.375} C_VEL
LIN {X 0,Y 380.756,Z 375.449,A -85,B 0,C 180,E1 -12736.926,E2 -12736.926} C_VEL
LIN {X 0,Y 379.894,Z 373.869,A -85,B 0,C 180,E1 -12739.334,E2 -12739.334} C_VEL
LIN {X 0,Y 379.294,Z 373.38,A -85,B 0,C 180,E1 -12741.101,E2 -12741.101} C_VEL
LIN {X 0,Y 378.335,Z 373.635,A -85,B 0,C 180,E1 -12743.528,E2 -12743.528} C_VEL
LIN {X 0,Y 376.994,Z 374.876,A -85,B 0,C 180,E1 -12745.995,E2 -12745.995} C_VEL
LIN {X 0,Y 375.322,Z 377.765,A -85,B 0,C 180,E1 -12749.63,E2 -12749.63} C_VEL
LIN {X 0,Y 374.089,Z 381.444,A -85,B 0,C 180,E1 -12753.2,E2 -12753.2} C_VEL
LIN {X 0,Y 373.478,Z 384.77,A -85,B 0,C 180,E1 -12755.896,E2 -12755.896} C_VEL
LIN {X 0,Y 379.645,Z 398.45,A -85,B 0,C 180,E1 -12757.763,E2 -12757.763} C_VEL
LIN {X 0,Y 382.978,Z 408.294,A -85,B 0,C 180,E1 -12758.994,E2 -12758.994} C_VEL
LIN {X 0,Y 383.735,Z 411.145,A -85,B 0,C 180,E1 -12759.337,E2 -12759.337} C_VEL
LIN {X 0,Y 382.024,Z 424.879,A -85,B 0,C 180,E1 -12760.499,E2 -12760.499} C_VEL
LIN {X 0,Y 380.182,Z 437.7,A -85,B 0,C 180,E1 -12761.824,E2 -12761.824} C_VEL
LIN {X 0,Y 378.473,Z 449.164,A -85,B 0,C 180,E1 -12763.273,E2 -12763.273} C_VEL
LIN {X 0,Y 376.84,Z 459.543,A -85,B 0,C 180,E1 -12764.865,E2 -12764.865} C_VEL
LIN {X 0,Y 375.446,Z 468.091,A -85,B 0,C 180,E1 -12766.468,E2 -12766.468} C_VEL
LIN {X 0,Y 374,Z 476.291,A -85,B 0,C 180,E1 -12768.346,E2 -12768.346} C_VEL
LIN {X 0,Y 372.694,Z 482.701,A -85,B 0,C 180,E1 -12770.229,E2 -12770.229} C_VEL
LIN {X 0,Y 371.855,Z 486.98,A -85,B 0,C 180,E1 -12771.851,E2 -12771.851} C_VEL
LIN {X 0,Y 371.168,Z 490.235,A -85,B 0,C 180,E1 -12773.477,E2 -12773.477} C_VEL
LIN {X 0,Y 370.909,Z 491.801,A -85,B 0,C 180,E1 -12774.564,E2 -12774.564} C_VEL
LIN {X 0,Y 370.537,Z 492.992,A -85,B 0,C 180,E1 -12775.649,E2 -12775.649} C_VEL
LIN {X 0,Y 370.244,Z 493.781,A -85,B 0,C 180,E1 -12776.736,E2 -12776.736} C_VEL
LIN {X 0,Y 369.935,Z 494.189,A -85,B 0,C 180,E1 -12777.823,E2 -12777.823} C_VEL
LIN {X 0,Y 369.766,Z 494.148,A -85,B 0,C 180,E1 -12778.911,E2 -12778.911} C_VEL
LIN {X 0,Y 369.603,Z 493.691,A -85,B 0,C 180,E1 -12780,E2 -12780} C_VEL
LIN {X 0,Y 369.503,Z 492.828,A -85,B 0,C 180,E1 -12781.09,E2 -12781.09} C_VEL
LIN {X 0,Y 369.446,Z 491.561,A -85,B 0,C 180,E1 -12782.181,E2 -12782.181} C_VEL
LIN {X 0,Y 369.538,Z 488.826,A -85,B 0,C 180,E1 -12783.817,E2 -12783.817} C_VEL
LIN {X 0,Y 369.449,Z 485.145,A -85,B 0,C 180,E1 -12785.458,E2 -12785.458} C_VEL
LIN {X 0,Y 369.917,Z 479.885,A -85,B 0,C 180,E1 -12787.234,E2 -12787.234} C_VEL
LIN {X 0,Y 370.348,Z 473.412,A -85,B 0,C 180,E1 -12788.985,E2 -12788.985} C_VEL
LIN {X 0,Y 370.834,Z 465.841,A -85,B 0,C 180,E1 -12790.649,E2 -12790.649} C_VEL
LIN {X 0,Y 371.475,Z 456.747,A -85,B 0,C 180,E1 -12792.289,E2 -12792.289} C_VEL
LIN {X 0,Y 372.102,Z 447.702,A -85,B 0,C 180,E1 -12793.656,E2 -12793.656} C_VEL
LIN {X 0,Y 373.043,Z 435.778,A -85,B 0,C 180,E1 -12795.154,E2 -12795.154} C_VEL
LIN {X 0,Y 373.873,Z 422.321,A -85,B 0,C 180,E1 -12796.521,E2 -12796.521} C_VEL
LIN {X 0,Y 374.848,Z 409.062,A -85,B 0,C 180,E1 -12797.598,E2 -12797.598} C_VEL
LIN {X 0,Y 375.451,Z 397.707,A -85,B 0,C 180,E1 -12798.344,E2 -12798.344} C_VEL
LIN {X 0,Y 372.089,Z 382.949,A -85,B 0,C 180,E1 -12799.3,E2 -12799.3} C_VEL
LIN {X 0,Y 368.86,Z 370.093,A -85,B 0,C 180,E1 -12799.985,E2 -12799.985} C_VEL
LIN {X 0,Y 369.074,Z 363.68,A -85,B 0,C 180,E1 -12803.572,E2 -12803.572} C_VEL
LIN {X 0,Y 369.293,Z 358.41,A -85,B 0,C 180,E1 -12806.558,E2 -12806.558} C_VEL
LIN {X 0,Y 369.561,Z 353.091,A -85,B 0,C 180,E1 -12809.634,E2 -12809.634} C_VEL
LIN {X 0,Y 369.788,Z 348.827,A -85,B 0,C 180,E1 -12812.152,E2 -12812.152} C_VEL
LIN {X 0,Y 369.981,Z 343.689,A -85,B 0,C 180,E1 -12815.231,E2 -12815.231} C_VEL
LIN {X 0,Y 369.775,Z 340.116,A -85,B 0,C 180,E1 -12817.46,E2 -12817.46} C_VEL
LIN {X 0,Y 368.949,Z 334.843,A -85,B 0,C 180,E1 -12820.904,E2 -12820.904} C_VEL
LIN {X 0,Y 368.889,Z 334.845,A -85,B 0,C 180,E1 -12824.823,E2 -12824.823} C_VEL
LIN {X 0,Y 368.922,Z 334.946,A -85,B 0,C 180,E1 -12828.277,E2 -12828.277} C_VEL
LIN {X 0,Y 370.241,Z 341.42,A -85,B 0,C 180,E1 -12831.212,E2 -12831.212} C_VEL
LIN {X 0,Y 371.08,Z 346.164,A -85,B 0,C 180,E1 -12833.413,E2 -12833.413} C_VEL
LIN {X 0,Y 371.278,Z 350.375,A -85,B 0,C 180,E1 -12835.395,E2 -12835.395} C_VEL
LIN {X 0,Y 371.092,Z 357.026,A -85,B 0,C 180,E1 -12838.457,E2 -12838.457} C_VEL
LIN {X 0,Y 370.97,Z 364.033,A -85,B 0,C 180,E1 -12841.728,E2 -12841.728} C_VEL
LIN {X 0,Y 370.968,Z 372.18,A -85,B 0,C 180,E1 -12845.418,E2 -12845.418} C_VEL
LIN {X 0,Y 371.119,Z 380.456,A -85,B 0,C 180,E1 -12848.909,E2 -12848.909} C_VEL
LIN {X 0,Y 371.265,Z 384.777,A -85,B 0,C 180,E1 -12850.547,E2 -12850.547} C_VEL
LIN {X 0,Y 375.218,Z 397.006,A -85,B 0,C 180,E1 -12851.147,E2 -12851.147} C_VEL
LIN {X 0,Y 376.428,Z 401.678,A -85,B 0,C 180,E1 -12851.416,E2 -12851.416} C_VEL
LIN {X 0,Y 375.958,Z 414.494,A -85,B 0,C 180,E1 -12852.11,E2 -12852.11} C_VEL
LIN {X 0,Y 375.383,Z 426.876,A -85,B 0,C 180,E1 -12853.026,E2 -12853.026} C_VEL
LIN {X 0,Y 374.63,Z 437.774,A -85,B 0,C 180,E1 -12854.074,E2 -12854.074} C_VEL
LIN {X 0,Y 373.645,Z 448.948,A -85,B 0,C 180,E1 -12855.427,E2 -12855.427} C_VEL
LIN {X 0,Y 372.931,Z 457.076,A -85,B 0,C 180,E1 -12856.65,E2 -12856.65} C_VEL
LIN {X 0,Y 371.961,Z 465.891,A -85,B 0,C 180,E1 -12858.278,E2 -12858.278} C_VEL
LIN {X 0,Y 371.301,Z 472.583,A -85,B 0,C 180,E1 -12859.823,E2 -12859.823} C_VEL
LIN {X 0,Y 370.794,Z 477.704,A -85,B 0,C 180,E1 -12861.276,E2 -12861.276} C_VEL
LIN {X 0,Y 369.967,Z 482.37,A -85,B 0,C 180,E1 -12862.905,E2 -12862.905} C_VEL
LIN {X 0,Y 369.621,Z 485.891,A -85,B 0,C 180,E1 -12864.542,E2 -12864.542} C_VEL
LIN {X 0,Y 369.535,Z 487.69,A -85,B 0,C 180,E1 -12865.635,E2 -12865.635} C_VEL
LIN {X 0,Y 369.446,Z 489.067,A -85,B 0,C 180,E1 -12866.726,E2 -12866.726} C_VEL
LIN {X 0,Y 369.133,Z 490.66,A -85,B 0,C 180,E1 -12868.906,E2 -12868.906} C_VEL
LIN {X 0,Y 369.092,Z 490.893,A -85,B 0,C 180,E1 -12869.997,E2 -12869.997} C_VEL
LIN {X 0,Y 369.25,Z 490.124,A -85,B 0,C 180,E1 -12872.179,E2 -12872.179} C_VEL
LIN {X 0,Y 369.454,Z 489.167,A -85,B 0,C 180,E1 -12873.269,E2 -12873.269} C_VEL
LIN {X 0,Y 369.572,Z 487.842,A -85,B 0,C 180,E1 -12874.36,E2 -12874.36} C_VEL
LIN {X 0,Y 369.783,Z 485.058,A -85,B 0,C 180,E1 -12875.997,E2 -12875.997} C_VEL
LIN {X 0,Y 370.268,Z 481.24,A -85,B 0,C 180,E1 -12877.632,E2 -12877.632} C_VEL
LIN {X 0,Y 370.953,Z 476.279,A -85,B 0,C 180,E1 -12879.264,E2 -12879.264} C_VEL
LIN {X 0,Y 371.53,Z 470.055,A -85,B 0,C 180,E1 -12880.901,E2 -12880.901} C_VEL
LIN {X 0,Y 372.391,Z 462.28,A -85,B 0,C 180,E1 -12882.532,E2 -12882.532} C_VEL
LIN {X 0,Y 373.265,Z 454.314,A -85,B 0,C 180,E1 -12883.887,E2 -12883.887} C_VEL
LIN {X 0,Y 374.01,Z 445.633,A -85,B 0,C 180,E1 -12885.11,E2 -12885.11} C_VEL
LIN {X 0,Y 374.795,Z 434.863,A -85,B 0,C 180,E1 -12886.333,E2 -12886.333} C_VEL
LIN {X 0,Y 375.575,Z 423.145,A -85,B 0,C 180,E1 -12887.379,E2 -12887.379} C_VEL
LIN {X 0,Y 376.182,Z 411.663,A -85,B 0,C 180,E1 -12888.162,E2 -12888.162} C_VEL
LIN {X 0,Y 376.402,Z 400.952,A -85,B 0,C 180,E1 -12888.719,E2 -12888.719} C_VEL
LIN {X 0,Y 372.414,Z 388.155,A -85,B 0,C 180,E1 -12889.404,E2 -12889.404} C_VEL
LIN {X 0,Y 371.398,Z 385.304,A -85,B 0,C 180,E1 -12889.536,E2 -12889.536} C_VEL
LIN {X 0,Y 370.676,Z 384.493,A -85,B 0,C 180,E1 -12889.692,E2 -12889.692} C_VEL
LIN {X 0,Y 368.881,Z 383.55,A -85,B 0,C 180,E1 -12890.259,E2 -12890.259} C_VEL
LIN {X 0,Y 366.296,Z 381.189,A -85,B 0,C 180,E1 -12891.536,E2 -12891.536} C_VEL
LIN {X 0,Y 365.575,Z 380.407,A -85,B 0,C 180,E1 -12892.052,E2 -12892.052} C_VEL
LIN {X 0,Y 364.347,Z 377.21,A -85,B 0,C 180,E1 -12893.402,E2 -12893.402} C_VEL
LIN {X 0,Y 364.152,Z 375.503,A -85,B 0,C 180,E1 -12894.081,E2 -12894.081} C_VEL
LIN {X 0,Y 364.106,Z 367.635,A -85,B 0,C 180,E1 -12897.593,E2 -12897.593} C_VEL
LIN {X 0,Y 364.212,Z 360.861,A -85,B 0,C 180,E1 -12900.75,E2 -12900.75} C_VEL
LIN {X 0,Y 364.387,Z 353.853,A -85,B 0,C 180,E1 -12904.005,E2 -12904.005} C_VEL
LIN {X 0,Y 364.218,Z 348.053,A -85,B 0,C 180,E1 -12906.735,E2 -12906.735} C_VEL
LIN {X 0,Y 363.078,Z 341.689,A -85,B 0,C 180,E1 -12909.696,E2 -12909.696} C_VEL
LIN {X 0,Y 361.829,Z 335.729,A -85,B 0,C 180,E1 -12912.43,E2 -12912.43} C_VEL
LIN {X 0,Y 361.884,Z 335.719,A -85,B 0,C 180,E1 -12915.931,E2 -12915.931} C_VEL
LIN {X 0,Y 361.89,Z 335.719,A -85,B 0,C 180,E1 -12919.229,E2 -12919.229} C_VEL
LIN {X 0,Y 361.857,Z 335.724,A -85,B 0,C 180,E1 -12922.98,E2 -12922.98} C_VEL
LIN {X 0,Y 361.84,Z 335.723,A -85,B 0,C 180,E1 -12926.628,E2 -12926.628} C_VEL
LIN {X 0,Y 361.855,Z 335.718,A -85,B 0,C 180,E1 -12929.67,E2 -12929.67} C_VEL
LIN {X 0,Y 361.934,Z 335.705,A -85,B 0,C 180,E1 -12933.473,E2 -12933.473} C_VEL
LIN {X 0,Y 361.902,Z 335.709,A -85,B 0,C 180,E1 -12937.145,E2 -12937.145} C_VEL
LIN {X 0,Y 361.913,Z 335.711,A -85,B 0,C 180,E1 -12940.723,E2 -12940.723} C_VEL
LIN {X 0,Y 361.924,Z 335.714,A -85,B 0,C 180,E1 -12944.225,E2 -12944.225} C_VEL
LIN {X 0,Y 361.978,Z 335.7,A -85,B 0,C 180,E1 -12946.527,E2 -12946.527} C_VEL
LIN {X 0,Y 362.015,Z 335.695,A -85,B 0,C 180,E1 -12949.937,E2 -12949.937} C_VEL
LIN {X 0,Y 362.128,Z 335.69,A -85,B 0,C 180,E1 -12952.192,E2 -12952.192} C_VEL
LIN {X 0,Y 362.094,Z 335.688,A -85,B 0,C 180,E1 -12954.43,E2 -12954.43} C_VEL
LIN {X 0,Y 362.255,Z 335.673,A -85,B 0,C 180,E1 -12957.776,E2 -12957.776} C_VEL
LIN {X 0,Y 362.402,Z 335.648,A -85,B 0,C 180,E1 -12960,E2 -12960} C_VEL
LIN {X 0,Y 362.267,Z 335.668,A -85,B 0,C 180,E1 -12962.223,E2 -12962.223} C_VEL
LIN {X 0,Y 362.154,Z 335.684,A -85,B 0,C 180,E1 -12966.686,E2 -12966.686} C_VEL
LIN {X 0,Y 362.051,Z 335.699,A -85,B 0,C 180,E1 -12968.933,E2 -12968.933} C_VEL
LIN {X 0,Y 361.943,Z 335.714,A -85,B 0,C 180,E1 -12972.332,E2 -12972.332} C_VEL
LIN {X 0,Y 361.94,Z 335.714,A -85,B 0,C 180,E1 -12974.621,E2 -12974.621} C_VEL
LIN {X 0,Y 361.938,Z 335.714,A -85,B 0,C 180,E1 -12978.1,E2 -12978.1} C_VEL
LIN {X 0,Y 361.909,Z 335.716,A -85,B 0,C 180,E1 -12981.651,E2 -12981.651} C_VEL
LIN {X 0,Y 361.908,Z 335.717,A -85,B 0,C 180,E1 -12985.291,E2 -12985.291} C_VEL
LIN {X 0,Y 361.891,Z 335.716,A -85,B 0,C 180,E1 -12987.78,E2 -12987.78} C_VEL
LIN {X 0,Y 361.825,Z 335.729,A -85,B 0,C 180,E1 -12991.287,E2 -12991.287} C_VEL
LIN {X 0,Y 361.845,Z 335.893,A -85,B 0,C 180,E1 -12994.027,E2 -12994.027} C_VEL
LIN {X 0,Y 364.384,Z 344.641,A -85,B 0,C 180,E1 -12997.466,E2 -12997.466} C_VEL
LIN {X 0,Y 367.488,Z 355.058,A -85,B 0,C 180,E1 -13001.237,E2 -13001.237} C_VEL
LIN {X 0,Y 371.298,Z 368.177,A -85,B 0,C 180,E1 -13005.551,E2 -13005.551} C_VEL
LIN {X 0,Y 374.188,Z 378.68,A -85,B 0,C 180,E1 -13008.701,E2 -13008.701} C_VEL
LIN {X 0,Y 375.935,Z 385.17,A -85,B 0,C 180,E1 -13010.538,E2 -13010.538} C_VEL
LIN {X 0,Y 376.133,Z 386.574,A -85,B 0,C 180,E1 -13010.909,E2 -13010.909} C_VEL
LIN {X 0,Y 373.799,Z 398.355,A -85,B 0,C 180,E1 -13013.615,E2 -13013.615} C_VEL
LIN {X 0,Y 370.804,Z 415.605,A -85,B 0,C 180,E1 -13017.466,E2 -13017.466} C_VEL
LIN {X 0,Y 375.102,Z 440.375,A -85,B 0,C 180,E1 -13018.496,E2 -13018.496} C_VEL
LIN {X 0,Y 377.612,Z 457.535,A -85,B 0,C 180,E1 -13019.405,E2 -13019.405} C_VEL
LIN {X 0,Y 378.264,Z 461.404,A -85,B 0,C 180,E1 -13019.644,E2 -13019.644} C_VEL
LIN {X 0,Y 376.67,Z 477.484,A -85,B 0,C 180,E1 -13020.524,E2 -13020.524} C_VEL
LIN {X 0,Y 374.789,Z 492.919,A -85,B 0,C 180,E1 -13021.59,E2 -13021.59} C_VEL
LIN {X 0,Y 372.947,Z 507.346,A -85,B 0,C 180,E1 -13022.819,E2 -13022.819} C_VEL
LIN {X 0,Y 370.92,Z 520.688,A -85,B 0,C 180,E1 -13024.168,E2 -13024.168} C_VEL
LIN {X 0,Y 368.857,Z 534.317,A -85,B 0,C 180,E1 -13025.821,E2 -13025.821} C_VEL
LIN {X 0,Y 366.803,Z 547.696,A -85,B 0,C 180,E1 -13027.768,E2 -13027.768} C_VEL
LIN {X 0,Y 365.081,Z 558.963,A -85,B 0,C 180,E1 -13029.729,E2 -13029.729} C_VEL
LIN {X 0,Y 363.689,Z 568.774,A -85,B 0,C 180,E1 -13031.746,E2 -13031.746} C_VEL
LIN {X 0,Y 362.533,Z 577.899,A -85,B 0,C 180,E1 -13033.967,E2 -13033.967} C_VEL
LIN {X 0,Y 361.701,Z 585.835,A -85,B 0,C 180,E1 -13036.292,E2 -13036.292} C_VEL
LIN {X 0,Y 361.097,Z 592.705,A -85,B 0,C 180,E1 -13038.78,E2 -13038.78} C_VEL
LIN {X 0,Y 360.824,Z 598.659,A -85,B 0,C 180,E1 -13041.603,E2 -13041.603} C_VEL
LIN {X 0,Y 360.823,Z 601.462,A -85,B 0,C 180,E1 -13043.391,E2 -13043.391} C_VEL
LIN {X 0,Y 360.797,Z 603.935,A -85,B 0,C 180,E1 -13045.534,E2 -13045.534} C_VEL
LIN {X 0,Y 360.895,Z 604.816,A -85,B 0,C 180,E1 -13046.654,E2 -13046.654} C_VEL
LIN {X 0,Y 360.807,Z 605.784,A -85,B 0,C 180,E1 -13048.887,E2 -13048.887} C_VEL
LIN {X 0,Y 360.823,Z 605.661,A -85,B 0,C 180,E1 -13051.119,E2 -13051.119} C_VEL
LIN {X 0,Y 360.901,Z 604.485,A -85,B 0,C 180,E1 -13053.352,E2 -13053.352} C_VEL
LIN {X 0,Y 360.82,Z 602.205,A -85,B 0,C 180,E1 -13055.591,E2 -13055.591} C_VEL
LIN {X 0,Y 360.931,Z 598.803,A -85,B 0,C 180,E1 -13057.837,E2 -13057.837} C_VEL
LIN {X 0,Y 360.997,Z 594.282,A -85,B 0,C 180,E1 -13060.094,E2 -13060.094} C_VEL
LIN {X 0,Y 361.413,Z 588.48,A -85,B 0,C 180,E1 -13062.354,E2 -13062.354} C_VEL
LIN {X 0,Y 362.028,Z 581.405,A -85,B 0,C 180,E1 -13064.62,E2 -13064.62} C_VEL
LIN {X 0,Y 362.999,Z 572.929,A -85,B 0,C 180,E1 -13066.885,E2 -13066.885} C_VEL
LIN {X 0,Y 364.218,Z 562.813,A -85,B 0,C 180,E1 -13069.152,E2 -13069.152} C_VEL
LIN {X 0,Y 365.952,Z 550.811,A -85,B 0,C 180,E1 -13071.403,E2 -13071.403} C_VEL
LIN {X 0,Y 367.934,Z 537.964,A -85,B 0,C 180,E1 -13073.427,E2 -13073.427} C_VEL
LIN {X 0,Y 369.947,Z 525.016,A -85,B 0,C 180,E1 -13075.157,E2 -13075.157} C_VEL
LIN {X 0,Y 372.213,Z 510.503,A -85,B 0,C 180,E1 -13076.797,E2 -13076.797} C_VEL
LIN {X 0,Y 374.378,Z 496.435,A -85,B 0,C 180,E1 -13078.129,E2 -13078.129} C_VEL
LIN {X 0,Y 376.266,Z 483.046,A -85,B 0,C 180,E1 -13079.209,E2 -13079.209} C_VEL
LIN {X 0,Y 378.416,Z 466.462,A -85,B 0,C 180,E1 -13080.302,E2 -13080.302} C_VEL
LIN {X 0,Y 378.89,Z 461.782,A -85,B 0,C 180,E1 -13080.567,E2 -13080.567} C_VEL
LIN {X 0,Y 377.379,Z 446.436,A -85,B 0,C 180,E1 -13081.628,E2 -13081.628} C_VEL
LIN {X 0,Y 376.271,Z 433.573,A -85,B 0,C 180,E1 -13082.382,E2 -13082.382} C_VEL
LIN {X 0,Y 373.995,Z 420.679,A -85,B 0,C 180,E1 -13083.174,E2 -13083.174} C_VEL
LIN {X 0,Y 372.034,Z 411.592,A -85,B 0,C 180,E1 -13083.807,E2 -13083.807} C_VEL
LIN {X 0,Y 375.377,Z 398.776,A -85,B 0,C 180,E1 -13087.145,E2 -13087.145} C_VEL
LIN {X 0,Y 377.847,Z 391.572,A -85,B 0,C 180,E1 -13089.23,E2 -13089.23} C_VEL
LIN {X 0,Y 377.951,Z 390.153,A -85,B 0,C 180,E1 -13089.733,E2 -13089.733} C_VEL
LIN {X 0,Y 376.898,Z 385.753,A -85,B 0,C 180,E1 -13091.766,E2 -13091.766} C_VEL
LIN {X 0,Y 375.812,Z 382.295,A -85,B 0,C 180,E1 -13093.785,E2 -13093.785} C_VEL
LIN {X 0,Y 374.729,Z 379.384,A -85,B 0,C 180,E1 -13096.058,E2 -13096.058} C_VEL
LIN {X 0,Y 373.65,Z 377.17,A -85,B 0,C 180,E1 -13098.829,E2 -13098.829} C_VEL
LIN {X 0,Y 372.657,Z 376.348,A -85,B 0,C 180,E1 -13101.512,E2 -13101.512} C_VEL
LIN {X 0,Y 372.175,Z 376.383,A -85,B 0,C 180,E1 -13102.824,E2 -13102.824} C_VEL
LIN {X 0,Y 370.805,Z 377.311,A -85,B 0,C 180,E1 -13105.348,E2 -13105.348} C_VEL
LIN {X 0,Y 368.92,Z 379.902,A -85,B 0,C 180,E1 -13109.046,E2 -13109.046} C_VEL
LIN {X 0,Y 367.569,Z 383.363,A -85,B 0,C 180,E1 -13112.685,E2 -13112.685} C_VEL
LIN {X 0,Y 366.927,Z 385.809,A -85,B 0,C 180,E1 -13114.903,E2 -13114.903} C_VEL
LIN {X 0,Y 368.247,Z 388.761,A -85,B 0,C 180,E1 -13115.352,E2 -13115.352} C_VEL
LIN {X 0,Y 373.022,Z 398.914,A -85,B 0,C 180,E1 -13116.882,E2 -13116.882} C_VEL
LIN {X 0,Y 376.981,Z 410.314,A -85,B 0,C 180,E1 -13118.418,E2 -13118.418} C_VEL
LIN {X 0,Y 377.876,Z 413.896,A -85,B 0,C 180,E1 -13118.876,E2 -13118.876} C_VEL
LIN {X 0,Y 375.849,Z 427.943,A -85,B 0,C 180,E1 -13120.115,E2 -13120.115} C_VEL
LIN {X 0,Y 373.852,Z 440.708,A -85,B 0,C 180,E1 -13121.505,E2 -13121.505} C_VEL
LIN {X 0,Y 372.047,Z 451.817,A -85,B 0,C 180,E1 -13122.975,E2 -13122.975} C_VEL
LIN {X 0,Y 370.302,Z 461.847,A -85,B 0,C 180,E1 -13124.591,E2 -13124.591} C_VEL
LIN {X 0,Y 368.779,Z 470.484,A -85,B 0,C 180,E1 -13126.275,E2 -13126.275} C_VEL
LIN {X 0,Y 367.312,Z 478.172,A -85,B 0,C 180,E1 -13128.131,E2 -13128.131} C_VEL
LIN {X 0,Y 365.913,Z 484.456,A -85,B 0,C 180,E1 -13130.046,E2 -13130.046} C_VEL
LIN {X 0,Y 365.014,Z 488.616,A -85,B 0,C 180,E1 -13131.698,E2 -13131.698} C_VEL
LIN {X 0,Y 364.287,Z 491.752,A -85,B 0,C 180,E1 -13133.353,E2 -13133.353} C_VEL
LIN {X 0,Y 363.995,Z 493.276,A -85,B 0,C 180,E1 -13134.46,E2 -13134.46} C_VEL
LIN {X 0,Y 363.622,Z 494.418,A -85,B 0,C 180,E1 -13135.566,E2 -13135.566} C_VEL
LIN {X 0,Y 363.301,Z 495.156,A -85,B 0,C 180,E1 -13136.673,E2 -13136.673} C_VEL
LIN {X 0,Y 362.963,Z 495.501,A -85,B 0,C 180,E1 -13137.781,E2 -13137.781} C_VEL
LIN {X 0,Y 362.779,Z 495.39,A -85,B 0,C 180,E1 -13138.89,E2 -13138.89} C_VEL
LIN {X 0,Y 362.624,Z 494.881,A -85,B 0,C 180,E1 -13140,E2 -13140} C_VEL
LIN {X 0,Y 362.498,Z 493.97,A -85,B 0,C 180,E1 -13141.111,E2 -13141.111} C_VEL
LIN {X 0,Y 362.446,Z 492.65,A -85,B 0,C 180,E1 -13142.223,E2 -13142.223} C_VEL
LIN {X 0,Y 362.543,Z 489.833,A -85,B 0,C 180,E1 -13143.891,E2 -13143.891} C_VEL
LIN {X 0,Y 362.442,Z 486.065,A -85,B 0,C 180,E1 -13145.564,E2 -13145.564} C_VEL
LIN {X 0,Y 362.916,Z 480.966,A -85,B 0,C 180,E1 -13147.295,E2 -13147.295} C_VEL
LIN {X 0,Y 363.374,Z 474.276,A -85,B 0,C 180,E1 -13149.124,E2 -13149.124} C_VEL
LIN {X 0,Y 363.879,Z 466.446,A -85,B 0,C 180,E1 -13150.855,E2 -13150.855} C_VEL
LIN {X 0,Y 364.551,Z 457.233,A -85,B 0,C 180,E1 -13152.526,E2 -13152.526} C_VEL
LIN {X 0,Y 365.34,Z 447.074,A -85,B 0,C 180,E1 -13154.056,E2 -13154.056} C_VEL
LIN {X 0,Y 366.186,Z 435.982,A -85,B 0,C 180,E1 -13155.444,E2 -13155.444} C_VEL
LIN {X 0,Y 367.062,Z 422.56,A -85,B 0,C 180,E1 -13156.819,E2 -13156.819} C_VEL
LIN {X 0,Y 368.081,Z 408.989,A -85,B 0,C 180,E1 -13157.927,E2 -13157.927} C_VEL
LIN {X 0,Y 368.465,Z 398.028,A -85,B 0,C 180,E1 -13158.667,E2 -13158.667} C_VEL
LIN {X 0,Y 364.837,Z 382.35,A -85,B 0,C 180,E1 -13159.701,E2 -13159.701} C_VEL
LIN {X 0,Y 361.848,Z 370.493,A -85,B 0,C 180,E1 -13160.345,E2 -13160.345} C_VEL
LIN {X 0,Y 362.054,Z 364.974,A -85,B 0,C 180,E1 -13163.45,E2 -13163.45} C_VEL
LIN {X 0,Y 362.292,Z 359.09,A -85,B 0,C 180,E1 -13166.828,E2 -13166.828} C_VEL
LIN {X 0,Y 362.595,Z 353.23,A -85,B 0,C 180,E1 -13170.262,E2 -13170.262} C_VEL
LIN {X 0,Y 362.916,Z 347.613,A -85,B 0,C 180,E1 -13173.619,E2 -13173.619} C_VEL
LIN {X 0,Y 363.016,Z 343.427,A -85,B 0,C 180,E1 -13176.191,E2 -13176.191} C_VEL
LIN {X 0,Y 362.415,Z 338.863,A -85,B 0,C 180,E1 -13179.13,E2 -13179.13} C_VEL
LIN {X 0,Y 361.852,Z 335.726,A -85,B 0,C 180,E1 -13181.328,E2 -13181.328} C_VEL
LIN {X 0,Y 361.826,Z 335.725,A -85,B 0,C 180,E1 -13184.368,E2 -13184.368} C_VEL
LIN {X 0,Y 361.844,Z 335.787,A -85,B 0,C 180,E1 -13187.728,E2 -13187.728} C_VEL
LIN {X 0,Y 363.195,Z 342.27,A -85,B 0,C 180,E1 -13190.717,E2 -13190.717} C_VEL
LIN {X 0,Y 364.169,Z 347.65,A -85,B 0,C 180,E1 -13193.252,E2 -13193.252} C_VEL
LIN {X 0,Y 364.419,Z 352.127,A -85,B 0,C 180,E1 -13195.323,E2 -13195.323} C_VEL
LIN {X 0,Y 364.215,Z 359.188,A -85,B 0,C 180,E1 -13198.598,E2 -13198.598} C_VEL
LIN {X 0,Y 364.088,Z 367.827,A -85,B 0,C 180,E1 -13202.616,E2 -13202.616} C_VEL
LIN {X 0,Y 364.147,Z 375.637,A -85,B 0,C 180,E1 -13206.088,E2 -13206.088} C_VEL
LIN {X 0,Y 364.27,Z 382.908,A -85,B 0,C 180,E1 -13209.086,E2 -13209.086} C_VEL
LIN {X 0,Y 364.36,Z 385.626,A -85,B 0,C 180,E1 -13210.144,E2 -13210.144} C_VEL
LIN {X 0,Y 368.674,Z 398.901,A -85,B 0,C 180,E1 -13210.837,E2 -13210.837} C_VEL
LIN {X 0,Y 369.766,Z 403.377,A -85,B 0,C 180,E1 -13211.101,E2 -13211.101} C_VEL
LIN {X 0,Y 369.291,Z 415.337,A -85,B 0,C 180,E1 -13211.762,E2 -13211.762} C_VEL
LIN {X 0,Y 368.677,Z 427.883,A -85,B 0,C 180,E1 -13212.703,E2 -13212.703} C_VEL
LIN {X 0,Y 367.893,Z 438.842,A -85,B 0,C 180,E1 -13213.774,E2 -13213.774} C_VEL
LIN {X 0,Y 366.858,Z 450.019,A -85,B 0,C 180,E1 -13215.151,E2 -13215.151} C_VEL
LIN {X 0,Y 366.118,Z 458.148,A -85,B 0,C 180,E1 -13216.397,E2 -13216.397} C_VEL
LIN {X 0,Y 365.23,Z 465.661,A -85,B 0,C 180,E1 -13217.777,E2 -13217.777} C_VEL
LIN {X 0,Y 364.567,Z 472.211,A -85,B 0,C 180,E1 -13219.252,E2 -13219.252} C_VEL
LIN {X 0,Y 363.868,Z 478.78,A -85,B 0,C 180,E1 -13221.109,E2 -13221.109} C_VEL
LIN {X 0,Y 363.004,Z 483.447,A -85,B 0,C 180,E1 -13222.768,E2 -13222.768} C_VEL
LIN {X 0,Y 362.637,Z 486.969,A -85,B 0,C 180,E1 -13224.437,E2 -13224.437} C_VEL
LIN {X 0,Y 362.536,Z 488.768,A -85,B 0,C 180,E1 -13225.55,E2 -13225.55} C_VEL
LIN {X 0,Y 362.443,Z 490.144,A -85,B 0,C 180,E1 -13226.662,E2 -13226.662} C_VEL
LIN {X 0,Y 362.117,Z 491.737,A -85,B 0,C 180,E1 -13228.885,E2 -13228.885} C_VEL
LIN {X 0,Y 362.075,Z 491.97,A -85,B 0,C 180,E1 -13229.997,E2 -13229.997} C_VEL
LIN {X 0,Y 362.238,Z 491.201,A -85,B 0,C 180,E1 -13232.221,E2 -13232.221} C_VEL
LIN {X 0,Y 362.451,Z 490.242,A -85,B 0,C 180,E1 -13233.332,E2 -13233.332} C_VEL
LIN {X 0,Y 362.594,Z 488.915,A -85,B 0,C 180,E1 -13234.444,E2 -13234.444} C_VEL
LIN {X 0,Y 362.801,Z 486.133,A -85,B 0,C 180,E1 -13236.113,E2 -13236.113} C_VEL
LIN {X 0,Y 363.315,Z 482.314,A -85,B 0,C 180,E1 -13237.779,E2 -13237.779} C_VEL
LIN {X 0,Y 364.036,Z 477.351,A -85,B 0,C 180,E1 -13239.442,E2 -13239.442} C_VEL
LIN {X 0,Y 364.741,Z 469.953,A -85,B 0,C 180,E1 -13241.388,E2 -13241.388} C_VEL
LIN {X 0,Y 365.54,Z 463.349,A -85,B 0,C 180,E1 -13242.771,E2 -13242.771} C_VEL
LIN {X 0,Y 366.453,Z 455.381,A -85,B 0,C 180,E1 -13244.151,E2 -13244.151} C_VEL
LIN {X 0,Y 367.242,Z 446.695,A -85,B 0,C 180,E1 -13245.395,E2 -13245.395} C_VEL
LIN {X 0,Y 368.068,Z 435.92,A -85,B 0,C 180,E1 -13246.64,E2 -13246.64} C_VEL
LIN {X 0,Y 368.808,Z 425.961,A -85,B 0,C 180,E1 -13247.557,E2 -13247.557} C_VEL
LIN {X 0,Y 369.438,Z 413.826,A -85,B 0,C 180,E1 -13248.434,E2 -13248.434} C_VEL
LIN {X 0,Y 369.685,Z 402.347,A -85,B 0,C 180,E1 -13249.056,E2 -13249.056} C_VEL
LIN {X 0,Y 365.746,Z 389.778,A -85,B 0,C 180,E1 -13249.755,E2 -13249.755} C_VEL
LIN {X 0,Y 364.388,Z 385.668,A -85,B 0,C 180,E1 -13249.949,E2 -13249.949} C_VEL
LIN {X 0,Y 364.185,Z 377.338,A -85,B 0,C 180,E1 -13253.3,E2 -13253.3} C_VEL
LIN {X 0,Y 364.152,Z 375.503,A -85,B 0,C 180,E1 -13254.081,E2 -13254.081} C_VEL
LIN {X 0,Y 363.453,Z 373.683,A -85,B 0,C 180,E1 -13254.957,E2 -13254.957} C_VEL
LIN {X 0,Y 360.616,Z 371.24,A -85,B 0,C 180,E1 -13256.409,E2 -13256.409} C_VEL
LIN {X 0,Y 358.278,Z 369.284,A -85,B 0,C 180,E1 -13257.588,E2 -13257.588} C_VEL
LIN {X 0,Y 357.335,Z 367.597,A -85,B 0,C 180,E1 -13258.489,E2 -13258.489} C_VEL
LIN {X 0,Y 357.288,Z 366.963,A -85,B 0,C 180,E1 -13258.791,E2 -13258.791} C_VEL
LIN {X 0,Y 357.423,Z 358.501,A -85,B 0,C 180,E1 -13262.747,E2 -13262.747} C_VEL
LIN {X 0,Y 357.531,Z 352.658,A -85,B 0,C 180,E1 -13265.438,E2 -13265.438} C_VEL
LIN {X 0,Y 357.094,Z 348.176,A -85,B 0,C 180,E1 -13267.593,E2 -13267.593} C_VEL
LIN {X 0,Y 355.848,Z 341.605,A -85,B 0,C 180,E1 -13270.669,E2 -13270.669} C_VEL
LIN {X 0,Y 354.801,Z 336.603,A -85,B 0,C 180,E1 -13272.947,E2 -13272.947} C_VEL
LIN {X 0,Y 354.826,Z 336.598,A -85,B 0,C 180,E1 -13276.112,E2 -13276.112} C_VEL
LIN {X 0,Y 354.841,Z 336.597,A -85,B 0,C 180,E1 -13279.186,E2 -13279.186} C_VEL
LIN {X 0,Y 354.797,Z 336.602,A -85,B 0,C 180,E1 -13282.399,E2 -13282.399} C_VEL
LIN {X 0,Y 354.795,Z 336.602,A -85,B 0,C 180,E1 -13284.938,E2 -13284.938} C_VEL
LIN {X 0,Y 354.774,Z 336.606,A -85,B 0,C 180,E1 -13288.403,E2 -13288.403} C_VEL
LIN {X 0,Y 354.829,Z 336.599,A -85,B 0,C 180,E1 -13291.617,E2 -13291.617} C_VEL
LIN {X 0,Y 354.88,Z 336.586,A -85,B 0,C 180,E1 -13294.171,E2 -13294.171} C_VEL
LIN {X 0,Y 354.871,Z 336.588,A -85,B 0,C 180,E1 -13297.896,E2 -13297.896} C_VEL
LIN {X 0,Y 354.902,Z 336.584,A -85,B 0,C 180,E1 -13301.889,E2 -13301.889} C_VEL
LIN {X 0,Y 354.92,Z 336.575,A -85,B 0,C 180,E1 -13305.98,E2 -13305.98} C_VEL
LIN {X 0,Y 354.962,Z 336.575,A -85,B 0,C 180,E1 -13309.735,E2 -13309.735} C_VEL
LIN {X 0,Y 355.091,Z 336.564,A -85,B 0,C 180,E1 -13312.036,E2 -13312.036} C_VEL
LIN {X 0,Y 355.068,Z 336.564,A -85,B 0,C 180,E1 -13314.32,E2 -13314.32} C_VEL
LIN {X 0,Y 355.218,Z 336.55,A -85,B 0,C 180,E1 -13317.732,E2 -13317.732} C_VEL
LIN {X 0,Y 355.351,Z 336.526,A -85,B 0,C 180,E1 -13320,E2 -13320} C_VEL
LIN {X 0,Y 355.231,Z 336.544,A -85,B 0,C 180,E1 -13322.267,E2 -13322.267} C_VEL
LIN {X 0,Y 355.119,Z 336.56,A -85,B 0,C 180,E1 -13326.819,E2 -13326.819} C_VEL
LIN {X 0,Y 354.993,Z 336.579,A -85,B 0,C 180,E1 -13329.112,E2 -13329.112} C_VEL
LIN {X 0,Y 354.903,Z 336.592,A -85,B 0,C 180,E1 -13332.581,E2 -13332.581} C_VEL
LIN {X 0,Y 354.868,Z 336.596,A -85,B 0,C 180,E1 -13336.096,E2 -13336.096} C_VEL
LIN {X 0,Y 354.887,Z 336.591,A -85,B 0,C 180,E1 -13338.472,E2 -13338.472} C_VEL
LIN {X 0,Y 354.869,Z 336.594,A -85,B 0,C 180,E1 -13342.103,E2 -13342.103} C_VEL
LIN {X 0,Y 354.877,Z 336.592,A -85,B 0,C 180,E1 -13345.829,E2 -13345.829} C_VEL
LIN {X 0,Y 354.832,Z 336.598,A -85,B 0,C 180,E1 -13349.68,E2 -13349.68} C_VEL
LIN {X 0,Y 354.807,Z 336.726,A -85,B 0,C 180,E1 -13353.09,E2 -13353.09} C_VEL
LIN {X 0,Y 357.027,Z 344.319,A -85,B 0,C 180,E1 -13356.195,E2 -13356.195} C_VEL
LIN {X 0,Y 359.506,Z 352.891,A -85,B 0,C 180,E1 -13359.445,E2 -13359.445} C_VEL
LIN {X 0,Y 362.192,Z 362.422,A -85,B 0,C 180,E1 -13362.776,E2 -13362.776} C_VEL
LIN {X 0,Y 365.303,Z 372.818,A -85,B 0,C 180,E1 -13366.169,E2 -13366.169} C_VEL
LIN {X 0,Y 368.325,Z 384.142,A -85,B 0,C 180,E1 -13369.557,E2 -13369.557} C_VEL
LIN {X 0,Y 369.327,Z 388.403,A -85,B 0,C 180,E1 -13370.753,E2 -13370.753} C_VEL
LIN {X 0,Y 366.547,Z 401.826,A -85,B 0,C 180,E1 -13373.886,E2 -13373.886} C_VEL
LIN {X 0,Y 364.128,Z 415.22,A -85,B 0,C 180,E1 -13376.949,E2 -13376.949} C_VEL
LIN {X 0,Y 368.295,Z 439.44,A -85,B 0,C 180,E1 -13377.989,E2 -13377.989} C_VEL
LIN {X 0,Y 370.81,Z 457.337,A -85,B 0,C 180,E1 -13378.952,E2 -13378.952} C_VEL
LIN {X 0,Y 371.575,Z 462.895,A -85,B 0,C 180,E1 -13379.295,E2 -13379.295} C_VEL
LIN {X 0,Y 369.888,Z 479.341,A -85,B 0,C 180,E1 -13380.243,E2 -13380.243} C_VEL
LIN {X 0,Y 367.943,Z 494.25,A -85,B 0,C 180,E1 -13381.324,E2 -13381.324} C_VEL
LIN {X 0,Y 366.051,Z 508.229,A -85,B 0,C 180,E1 -13382.566,E2 -13382.566} C_VEL
LIN {X 0,Y 363.817,Z 522.55,A -85,B 0,C 180,E1 -13384.087,E2 -13384.087} C_VEL
LIN {X 0,Y 361.888,Z 534.759,A -85,B 0,C 180,E1 -13385.63,E2 -13385.63} C_VEL
LIN {X 0,Y 360.031,Z 546.172,A -85,B 0,C 180,E1 -13387.327,E2 -13387.327} C_VEL
LIN {X 0,Y 358.241,Z 557.56,A -85,B 0,C 180,E1 -13389.325,E2 -13389.325} C_VEL
LIN {X 0,Y 356.888,Z 566.799,A -85,B 0,C 180,E1 -13391.227,E2 -13391.227} C_VEL
LIN {X 0,Y 355.77,Z 575.651,A -85,B 0,C 180,E1 -13393.358,E2 -13393.358} C_VEL
LIN {X 0,Y 354.765,Z 583.785,A -85,B 0,C 180,E1 -13395.724,E2 -13395.724} C_VEL
LIN {X 0,Y 354.208,Z 590.13,A -85,B 0,C 180,E1 -13397.978,E2 -13397.978} C_VEL
LIN {X 0,Y 353.825,Z 595.395,A -85,B 0,C 180,E1 -13400.283,E2 -13400.283} C_VEL
LIN {X 0,Y 353.79,Z 598.534,A -85,B 0,C 180,E1 -13402.01,E2 -13402.01} C_VEL
LIN {X 0,Y 353.698,Z 601.752,A -85,B 0,C 180,E1 -13404.301,E2 -13404.301} C_VEL
LIN {X 0,Y 353.865,Z 603.794,A -85,B 0,C 180,E1 -13406.587,E2 -13406.587} C_VEL
LIN {X 0,Y 353.777,Z 604.776,A -85,B 0,C 180,E1 -13408.865,E2 -13408.865} C_VEL
LIN {X 0,Y 353.794,Z 604.646,A -85,B 0,C 180,E1 -13411.141,E2 -13411.141} C_VEL
LIN {X 0,Y 353.873,Z 603.47,A -85,B 0,C 180,E1 -13413.418,E2 -13413.418} C_VEL
LIN {X 0,Y 353.775,Z 601.175,A -85,B 0,C 180,E1 -13415.703,E2 -13415.703} C_VEL
LIN {X 0,Y 353.876,Z 597.764,A -85,B 0,C 180,E1 -13417.994,E2 -13417.994} C_VEL
LIN {X 0,Y 353.964,Z 593.23,A -85,B 0,C 180,E1 -13420.296,E2 -13420.296} C_VEL
LIN {X 0,Y 354.378,Z 587.417,A -85,B 0,C 180,E1 -13422.603,E2 -13422.603} C_VEL
LIN {X 0,Y 355.02,Z 580.336,A -85,B 0,C 180,E1 -13424.915,E2 -13424.915} C_VEL
LIN {X 0,Y 356.065,Z 571.873,A -85,B 0,C 180,E1 -13427.224,E2 -13427.224} C_VEL
LIN {X 0,Y 357.355,Z 561.772,A -85,B 0,C 180,E1 -13429.534,E2 -13429.534} C_VEL
LIN {X 0,Y 359.178,Z 549.809,A -85,B 0,C 180,E1 -13431.827,E2 -13431.827} C_VEL
LIN {X 0,Y 361.317,Z 536.871,A -85,B 0,C 180,E1 -13433.909,E2 -13433.909} C_VEL
LIN {X 0,Y 363.565,Z 523.088,A -85,B 0,C 180,E1 -13435.784,E2 -13435.784} C_VEL
LIN {X 0,Y 366.018,Z 508.535,A -85,B 0,C 180,E1 -13437.443,E2 -13437.443} C_VEL
LIN {X 0,Y 368.491,Z 492.742,A -85,B 0,C 180,E1 -13438.947,E2 -13438.947} C_VEL
LIN {X 0,Y 370.841,Z 477.269,A -85,B 0,C 180,E1 -13440.149,E2 -13440.149} C_VEL
LIN {X 0,Y 372.635,Z 464.014,A -85,B 0,C 180,E1 -13441.006,E2 -13441.006} C_VEL
LIN {X 0,Y 371.511,Z 448.666,A -85,B 0,C 180,E1 -13442.13,E2 -13442.13} C_VEL
LIN {X 0,Y 370.386,Z 434.049,A -85,B 0,C 180,E1 -13443.048,E2 -13443.048} C_VEL
LIN {X 0,Y 368.121,Z 420.831,A -85,B 0,C 180,E1 -13443.934,E2 -13443.934} C_VEL
LIN {X 0,Y 365.924,Z 410.931,A -85,B 0,C 180,E1 -13444.683,E2 -13444.683} C_VEL
LIN {X 0,Y 368.959,Z 400.329,A -85,B 0,C 180,E1 -13447.559,E2 -13447.559} C_VEL
LIN {X 0,Y 371.185,Z 394.226,A -85,B 0,C 180,E1 -13449.371,E2 -13449.371} C_VEL
LIN {X 0,Y 371.344,Z 392.397,A -85,B 0,C 180,E1 -13450.054,E2 -13450.054} C_VEL
LIN {X 0,Y 370.282,Z 387.883,A -85,B 0,C 180,E1 -13452.25,E2 -13452.25} C_VEL
LIN {X 0,Y 368.902,Z 383.942,A -85,B 0,C 180,E1 -13454.823,E2 -13454.823} C_VEL
LIN {X 0,Y 368.123,Z 381.955,A -85,B 0,C 180,E1 -13456.584,E2 -13456.584} C_VEL
LIN {X 0,Y 367.449,Z 380.594,A -85,B 0,C 180,E1 -13458.242,E2 -13458.242} C_VEL
LIN {X 0,Y 366.52,Z 379.467,A -85,B 0,C 180,E1 -13460.745,E2 -13460.745} C_VEL
LIN {X 0,Y 365.982,Z 379.315,A -85,B 0,C 180,E1 -13462.085,E2 -13462.085} C_VEL
LIN {X 0,Y 365.071,Z 379.606,A -85,B 0,C 180,E1 -13463.957,E2 -13463.957} C_VEL
LIN {X 0,Y 363.187,Z 381.247,A -85,B 0,C 180,E1 -13467.193,E2 -13467.193} C_VEL
LIN {X 0,Y 361.49,Z 384.324,A -85,B 0,C 180,E1 -13471.034,E2 -13471.034} C_VEL
LIN {X 0,Y 360.567,Z 387.16,A -85,B 0,C 180,E1 -13473.844,E2 -13473.844} C_VEL
LIN {X 0,Y 365.793,Z 398.045,A -85,B 0,C 180,E1 -13475.693,E2 -13475.693} C_VEL
LIN {X 0,Y 369.438,Z 407.309,A -85,B 0,C 180,E1 -13477.093,E2 -13477.093} C_VEL
LIN {X 0,Y 371.924,Z 415.867,A -85,B 0,C 180,E1 -13478.291,E2 -13478.291} C_VEL
LIN {X 0,Y 369.912,Z 429.848,A -85,B 0,C 180,E1 -13479.591,E2 -13479.591} C_VEL
LIN {X 0,Y 367.539,Z 443.811,A -85,B 0,C 180,E1 -13481.175,E2 -13481.175} C_VEL
LIN {X 0,Y 365.655,Z 454.463,A -85,B 0,C 180,E1 -13482.668,E2 -13482.668} C_VEL
LIN {X 0,Y 363.803,Z 464.256,A -85,B 0,C 180,E1 -13484.309,E2 -13484.309} C_VEL
LIN {X 0,Y 362.28,Z 472.205,A -85,B 0,C 180,E1 -13485.929,E2 -13485.929} C_VEL
LIN {X 0,Y 360.83,Z 479.139,A -85,B 0,C 180,E1 -13487.629,E2 -13487.629} C_VEL
LIN {X 0,Y 359.577,Z 484.656,A -85,B 0,C 180,E1 -13489.3,E2 -13489.3} C_VEL
LIN {X 0,Y 358.436,Z 489.063,A -85,B 0,C 180,E1 -13490.976,E2 -13490.976} C_VEL
LIN {X 0,Y 357.848,Z 491.431,A -85,B 0,C 180,E1 -13492.099,E2 -13492.099} C_VEL
LIN {X 0,Y 357.423,Z 493.307,A -85,B 0,C 180,E1 -13493.225,E2 -13493.225} C_VEL
LIN {X 0,Y 357.1,Z 494.759,A -85,B 0,C 180,E1 -13494.353,E2 -13494.353} C_VEL
LIN {X 0,Y 356.369,Z 496.527,A -85,B 0,C 180,E1 -13496.609,E2 -13496.609} C_VEL
LIN {X 0,Y 356.007,Z 496.804,A -85,B 0,C 180,E1 -13497.738,E2 -13497.738} C_VEL
LIN {X 0,Y 355.792,Z 496.642,A -85,B 0,C 180,E1 -13498.869,E2 -13498.869} C_VEL
LIN {X 0,Y 355.639,Z 496.075,A -85,B 0,C 180,E1 -13500,E2 -13500} C_VEL
LIN {X 0,Y 355.513,Z 495.109,A -85,B 0,C 180,E1 -13501.133,E2 -13501.133} C_VEL
LIN {X 0,Y 355.444,Z 493.738,A -85,B 0,C 180,E1 -13502.267,E2 -13502.267} C_VEL
LIN {X 0,Y 355.543,Z 490.824,A -85,B 0,C 180,E1 -13503.968,E2 -13503.968} C_VEL
LIN {X 0,Y 355.433,Z 486.961,A -85,B 0,C 180,E1 -13505.674,E2 -13505.674} C_VEL
LIN {X 0,Y 355.923,Z 481.977,A -85,B 0,C 180,E1 -13507.375,E2 -13507.375} C_VEL
LIN {X 0,Y 356.4,Z 475.105,A -85,B 0,C 180,E1 -13509.268,E2 -13509.268} C_VEL
LIN {X 0,Y 356.93,Z 467.007,A -85,B 0,C 180,E1 -13511.069,E2 -13511.069} C_VEL
LIN {X 0,Y 357.643,Z 457.697,A -85,B 0,C 180,E1 -13512.772,E2 -13512.772} C_VEL
LIN {X 0,Y 358.464,Z 447.428,A -85,B 0,C 180,E1 -13514.331,E2 -13514.331} C_VEL
LIN {X 0,Y 359.328,Z 436.178,A -85,B 0,C 180,E1 -13515.747,E2 -13515.747} C_VEL
LIN {X 0,Y 360.264,Z 422.458,A -85,B 0,C 180,E1 -13517.161,E2 -13517.161} C_VEL
LIN {X 0,Y 361.309,Z 408.942,A -85,B 0,C 180,E1 -13518.266,E2 -13518.266} C_VEL
LIN {X 0,Y 361.702,Z 399.643,A -85,B 0,C 180,E1 -13518.908,E2 -13518.908} C_VEL
LIN {X 0,Y 358.246,Z 384.416,A -85,B 0,C 180,E1 -13519.951,E2 -13519.951} C_VEL
LIN {X 0,Y 354.844,Z 370.899,A -85,B 0,C 180,E1 -13520.712,E2 -13520.712} C_VEL
LIN {X 0,Y 355.036,Z 366.289,A -85,B 0,C 180,E1 -13523.323,E2 -13523.323} C_VEL
LIN {X 0,Y 355.299,Z 359.857,A -85,B 0,C 180,E1 -13527.062,E2 -13527.062} C_VEL
LIN {X 0,Y 355.6,Z 354.439,A -85,B 0,C 180,E1 -13530.264,E2 -13530.264} C_VEL
LIN {X 0,Y 355.908,Z 348.969,A -85,B 0,C 180,E1 -13533.567,E2 -13533.567} C_VEL
LIN {X 0,Y 356.039,Z 344.556,A -85,B 0,C 180,E1 -13536.313,E2 -13536.313} C_VEL
LIN {X 0,Y 355.367,Z 339.628,A -85,B 0,C 180,E1 -13539.527,E2 -13539.527} C_VEL
LIN {X 0,Y 354.805,Z 336.604,A -85,B 0,C 180,E1 -13541.712,E2 -13541.712} C_VEL
LIN {X 0,Y 354.773,Z 336.607,A -85,B 0,C 180,E1 -13545.493,E2 -13545.493} C_VEL
LIN {X 0,Y 354.827,Z 336.742,A -85,B 0,C 180,E1 -13547.236,E2 -13547.236} C_VEL
LIN {X 0,Y 356.223,Z 343.421,A -85,B 0,C 180,E1 -13550.304,E2 -13550.304} C_VEL
LIN {X 0,Y 357.32,Z 349.37,A -85,B 0,C 180,E1 -13553.136,E2 -13553.136} C_VEL
LIN {X 0,Y 357.557,Z 353.836,A -85,B 0,C 180,E1 -13555.246,E2 -13555.246} C_VEL
LIN {X 0,Y 357.344,Z 361.002,A -85,B 0,C 180,E1 -13558.586,E2 -13558.586} C_VEL
LIN {X 0,Y 357.216,Z 369.039,A -85,B 0,C 180,E1 -13562.295,E2 -13562.295} C_VEL
LIN {X 0,Y 357.316,Z 377.892,A -85,B 0,C 180,E1 -13566.218,E2 -13566.218} C_VEL
LIN {X 0,Y 357.502,Z 386.6,A -85,B 0,C 180,E1 -13569.735,E2 -13569.735} C_VEL
LIN {X 0,Y 362.176,Z 400.883,A -85,B 0,C 180,E1 -13570.522,E2 -13570.522} C_VEL
LIN {X 0,Y 363.098,Z 404.614,A -85,B 0,C 180,E1 -13570.75,E2 -13570.75} C_VEL
LIN {X 0,Y 362.634,Z 416.767,A -85,B 0,C 180,E1 -13571.441,E2 -13571.441} C_VEL
LIN {X 0,Y 361.983,Z 428.875,A -85,B 0,C 180,E1 -13572.366,E2 -13572.366} C_VEL
LIN {X 0,Y 361.162,Z 439.91,A -85,B 0,C 180,E1 -13573.463,E2 -13573.463} C_VEL
LIN {X 0,Y 360.079,Z 451.091,A -85,B 0,C 180,E1 -13574.865,E2 -13574.865} C_VEL
LIN {X 0,Y 359.308,Z 459.22,A -85,B 0,C 180,E1 -13576.134,E2 -13576.134} C_VEL
LIN {X 0,Y 358.381,Z 466.735,A -85,B 0,C 180,E1 -13577.54,E2 -13577.54} C_VEL
LIN {X 0,Y 357.702,Z 473.22,A -85,B 0,C 180,E1 -13579.027,E2 -13579.027} C_VEL
LIN {X 0,Y 356.944,Z 479.855,A -85,B 0,C 180,E1 -13580.935,E2 -13580.935} C_VEL
LIN {X 0,Y 356.044,Z 484.524,A -85,B 0,C 180,E1 -13582.626,E2 -13582.626} C_VEL
LIN {X 0,Y 355.653,Z 488.046,A -85,B 0,C 180,E1 -13584.327,E2 -13584.327} C_VEL
LIN {X 0,Y 355.564,Z 489.841,A -85,B 0,C 180,E1 -13585.463,E2 -13585.463} C_VEL
LIN {X 0,Y 355.438,Z 491.221,A -85,B 0,C 180,E1 -13586.597,E2 -13586.597} C_VEL
LIN {X 0,Y 355.102,Z 492.814,A -85,B 0,C 180,E1 -13588.863,E2 -13588.863} C_VEL
LIN {X 0,Y 355.058,Z 493.047,A -85,B 0,C 180,E1 -13589.997,E2 -13589.997} C_VEL
LIN {X 0,Y 355.226,Z 492.277,A -85,B 0,C 180,E1 -13592.265,E2 -13592.265} C_VEL
LIN {X 0,Y 355.449,Z 491.318,A -85,B 0,C 180,E1 -13593.398,E2 -13593.398} C_VEL
LIN {X 0,Y 355.613,Z 489.988,A -85,B 0,C 180,E1 -13594.531,E2 -13594.531} C_VEL
LIN {X 0,Y 355.822,Z 487.209,A -85,B 0,C 180,E1 -13596.234,E2 -13596.234} C_VEL
LIN {X 0,Y 356.364,Z 483.388,A -85,B 0,C 180,E1 -13597.932,E2 -13597.932} C_VEL
LIN {X 0,Y 357.122,Z 478.423,A -85,B 0,C 180,E1 -13599.626,E2 -13599.626} C_VEL
LIN {X 0,Y 357.864,Z 471.024,A -85,B 0,C 180,E1 -13601.61,E2 -13601.61} C_VEL
LIN {X 0,Y 358.91,Z 462.959,A -85,B 0,C 180,E1 -13603.299,E2 -13603.299} C_VEL
LIN {X 0,Y 359.764,Z 454.654,A -85,B 0,C 180,E1 -13604.709,E2 -13604.709} C_VEL
LIN {X 0,Y 360.793,Z 444.411,A -85,B 0,C 180,E1 -13606.113,E2 -13606.113} C_VEL
LIN {X 0,Y 361.575,Z 435.155,A -85,B 0,C 180,E1 -13607.142,E2 -13607.142} C_VEL
LIN {X 0,Y 362.235,Z 424.764,A -85,B 0,C 180,E1 -13608.082,E2 -13608.082} C_VEL
LIN {X 0,Y 362.887,Z 412.577,A -85,B 0,C 180,E1 -13608.922,E2 -13608.922} C_VEL
LIN {X 0,Y 363.118,Z 404.301,A -85,B 0,C 180,E1 -13609.368,E2 -13609.368} C_VEL
LIN {X 0,Y 359.405,Z 392.189,A -85,B 0,C 180,E1 -13610.076,E2 -13610.076} C_VEL
LIN {X 0,Y 357.552,Z 386.643,A -85,B 0,C 180,E1 -13610.361,E2 -13610.361} C_VEL
LIN {X 0,Y 357.329,Z 378.19,A -85,B 0,C 180,E1 -13613.775,E2 -13613.775} C_VEL
LIN {X 0,Y 357.258,Z 371.106,A -85,B 0,C 180,E1 -13616.898,E2 -13616.898} C_VEL
LIN {X 0,Y 357.288,Z 366.963,A -85,B 0,C 180,E1 -13618.791,E2 -13618.791} C_VEL
LIN {X 0,Y 356.725,Z 365.225,A -85,B 0,C 180,E1 -13619.691,E2 -13619.691} C_VEL
LIN {X 0,Y 354.021,Z 362.862,A -85,B 0,C 180,E1 -13621.181,E2 -13621.181} C_VEL
LIN {X 0,Y 351.702,Z 360.978,A -85,B 0,C 180,E1 -13622.386,E2 -13622.386} C_VEL
LIN {X 0,Y 350.721,Z 359.284,A -85,B 0,C 180,E1 -13623.304,E2 -13623.304} C_VEL
LIN {X 0,Y 350.65,Z 358.63,A -85,B 0,C 180,E1 -13623.61,E2 -13623.61} C_VEL
LIN {X 0,Y 350.669,Z 353.219,A -85,B 0,C 180,E1 -13626.096,E2 -13626.096} C_VEL
LIN {X 0,Y 349.979,Z 348.266,A -85,B 0,C 180,E1 -13628.496,E2 -13628.496} C_VEL
LIN {X 0,Y 348.594,Z 341.335,A -85,B 0,C 180,E1 -13631.758,E2 -13631.758} C_VEL
LIN {X 0,Y 347.735,Z 337.484,A -85,B 0,C 180,E1 -13633.601,E2 -13633.601} C_VEL
LIN {X 0,Y 347.769,Z 337.48,A -85,B 0,C 180,E1 -13636.673,E2 -13636.673} C_VEL
LIN {X 0,Y 347.77,Z 337.477,A -85,B 0,C 180,E1 -13640.163,E2 -13640.163} C_VEL
LIN {X 0,Y 347.773,Z 337.475,A -85,B 0,C 180,E1 -13644.122,E2 -13644.122} C_VEL
LIN {X 0,Y 347.72,Z 337.485,A -85,B 0,C 180,E1 -13648.084,E2 -13648.084} C_VEL
LIN {X 0,Y 347.785,Z 337.474,A -85,B 0,C 180,E1 -13650.988,E2 -13650.988} C_VEL
LIN {X 0,Y 347.811,Z 337.464,A -85,B 0,C 180,E1 -13653.606,E2 -13653.606} C_VEL
LIN {X 0,Y 347.797,Z 337.471,A -85,B 0,C 180,E1 -13656.162,E2 -13656.162} C_VEL
LIN {X 0,Y 347.822,Z 337.469,A -85,B 0,C 180,E1 -13659.909,E2 -13659.909} C_VEL
LIN {X 0,Y 347.845,Z 337.465,A -85,B 0,C 180,E1 -13662.358,E2 -13662.358} C_VEL
LIN {X 0,Y 347.875,Z 337.452,A -85,B 0,C 180,E1 -13665.969,E2 -13665.969} C_VEL
LIN {X 0,Y 347.912,Z 337.455,A -85,B 0,C 180,E1 -13669.525,E2 -13669.525} C_VEL
LIN {X 0,Y 348.051,Z 337.438,A -85,B 0,C 180,E1 -13671.874,E2 -13671.874} C_VEL
LIN {X 0,Y 348.044,Z 337.439,A -85,B 0,C 180,E1 -13674.205,E2 -13674.205} C_VEL
LIN {X 0,Y 348.181,Z 337.427,A -85,B 0,C 180,E1 -13677.686,E2 -13677.686} C_VEL
LIN {X 0,Y 348.301,Z 337.403,A -85,B 0,C 180,E1 -13680,E2 -13680} C_VEL
LIN {X 0,Y 348.194,Z 337.421,A -85,B 0,C 180,E1 -13682.313,E2 -13682.313} C_VEL
LIN {X 0,Y 348.086,Z 337.436,A -85,B 0,C 180,E1 -13686.958,E2 -13686.958} C_VEL
LIN {X 0,Y 347.945,Z 337.457,A -85,B 0,C 180,E1 -13689.299,E2 -13689.299} C_VEL
LIN {X 0,Y 347.87,Z 337.466,A -85,B 0,C 180,E1 -13692.84,E2 -13692.84} C_VEL
LIN {X 0,Y 347.818,Z 337.472,A -85,B 0,C 180,E1 -13696.432,E2 -13696.432} C_VEL
LIN {X 0,Y 347.84,Z 337.469,A -85,B 0,C 180,E1 -13698.861,E2 -13698.861} C_VEL
LIN {X 0,Y 347.817,Z 337.472,A -85,B 0,C 180,E1 -13702.576,E2 -13702.576} C_VEL
LIN {X 0,Y 347.809,Z 337.471,A -85,B 0,C 180,E1 -13706.394,E2 -13706.394} C_VEL
LIN {X 0,Y 347.787,Z 337.476,A -85,B 0,C 180,E1 -13709.673,E2 -13709.673} C_VEL
LIN {X 0,Y 347.732,Z 337.56,A -85,B 0,C 180,E1 -13712.124,E2 -13712.124} C_VEL
LIN {X 0,Y 350.45,Z 346.832,A -85,B 0,C 180,E1 -13716.018,E2 -13716.018} C_VEL
LIN {X 0,Y 353.097,Z 356.079,A -85,B 0,C 180,E1 -13719.562,E2 -13719.562} C_VEL
LIN {X 0,Y 355.861,Z 365.983,A -85,B 0,C 180,E1 -13723.058,E2 -13723.058} C_VEL
LIN {X 0,Y 358.613,Z 375.094,A -85,B 0,C 180,E1 -13726.072,E2 -13726.072} C_VEL
LIN {X 0,Y 361.751,Z 386.859,A -85,B 0,C 180,E1 -13729.644,E2 -13729.644} C_VEL
LIN {X 0,Y 362.443,Z 390.412,A -85,B 0,C 180,E1 -13730.652,E2 -13730.652} C_VEL
LIN {X 0,Y 359.112,Z 406.161,A -85,B 0,C 180,E1 -13734.397,E2 -13734.397} C_VEL
LIN {X 0,Y 357.442,Z 415.118,A -85,B 0,C 180,E1 -13736.457,E2 -13736.457} C_VEL
LIN {X 0,Y 361.458,Z 438.453,A -85,B 0,C 180,E1 -13737.467,E2 -13737.467} C_VEL
LIN {X 0,Y 363.781,Z 455.414,A -85,B 0,C 180,E1 -13738.381,E2 -13738.381} C_VEL
LIN {X 0,Y 364.905,Z 463.423,A -85,B 0,C 180,E1 -13738.897,E2 -13738.897} C_VEL
LIN {X 0,Y 363.329,Z 478.811,A -85,B 0,C 180,E1 -13739.81,E2 -13739.81} C_VEL
LIN {X 0,Y 361.315,Z 493.661,A -85,B 0,C 180,E1 -13740.907,E2 -13740.907} C_VEL
LIN {X 0,Y 359.396,Z 507.616,A -85,B 0,C 180,E1 -13742.172,E2 -13742.172} C_VEL
LIN {X 0,Y 357.076,Z 521.907,A -85,B 0,C 180,E1 -13743.718,E2 -13743.718} C_VEL
LIN {X 0,Y 354.904,Z 535.091,A -85,B 0,C 180,E1 -13745.431,E2 -13745.431} C_VEL
LIN {X 0,Y 353.026,Z 546.411,A -85,B 0,C 180,E1 -13747.161,E2 -13747.161} C_VEL
LIN {X 0,Y 351.202,Z 557.644,A -85,B 0,C 180,E1 -13749.198,E2 -13749.198} C_VEL
LIN {X 0,Y 349.767,Z 567.224,A -85,B 0,C 180,E1 -13751.25,E2 -13751.25} C_VEL
LIN {X 0,Y 348.541,Z 576.487,A -85,B 0,C 180,E1 -13753.606,E2 -13753.606} C_VEL
LIN {X 0,Y 347.622,Z 584.363,A -85,B 0,C 180,E1 -13756.031,E2 -13756.031} C_VEL
LIN {X 0,Y 347.062,Z 590.438,A -85,B 0,C 180,E1 -13758.32,E2 -13758.32} C_VEL
LIN {X 0,Y 346.746,Z 595.393,A -85,B 0,C 180,E1 -13760.672,E2 -13760.672} C_VEL
LIN {X 0,Y 346.753,Z 599.558,A -85,B 0,C 180,E1 -13763.278,E2 -13763.278} C_VEL
LIN {X 0,Y 346.729,Z 601.852,A -85,B 0,C 180,E1 -13765.352,E2 -13765.352} C_VEL
LIN {X 0,Y 346.836,Z 602.758,A -85,B 0,C 180,E1 -13766.518,E2 -13766.518} C_VEL
LIN {X 0,Y 346.749,Z 603.755,A -85,B 0,C 180,E1 -13768.841,E2 -13768.841} C_VEL
LIN {X 0,Y 346.765,Z 603.623,A -85,B 0,C 180,E1 -13771.164,E2 -13771.164} C_VEL
LIN {X 0,Y 346.846,Z 602.454,A -85,B 0,C 180,E1 -13773.488,E2 -13773.488} C_VEL
LIN {X 0,Y 346.73,Z 600.145,A -85,B 0,C 180,E1 -13775.819,E2 -13775.819} C_VEL
LIN {X 0,Y 346.819,Z 596.73,A -85,B 0,C 180,E1 -13778.158,E2 -13778.158} C_VEL
LIN {X 0,Y 346.92,Z 592.186,A -85,B 0,C 180,E1 -13780.508,E2 -13780.508} C_VEL
LIN {X 0,Y 347.351,Z 586.373,A -85,B 0,C 180,E1 -13782.862,E2 -13782.862} C_VEL
LIN {X 0,Y 348.033,Z 579.298,A -85,B 0,C 180,E1 -13785.222,E2 -13785.222} C_VEL
LIN {X 0,Y 349.082,Z 570.848,A -85,B 0,C 180,E1 -13787.58,E2 -13787.58} C_VEL
LIN {X 0,Y 350.542,Z 560.784,A -85,B 0,C 180,E1 -13789.93,E2 -13789.93} C_VEL
LIN {X 0,Y 352.412,Z 548.871,A -85,B 0,C 180,E1 -13792.269,E2 -13792.269} C_VEL
LIN {X 0,Y 354.683,Z 535.953,A -85,B 0,C 180,E1 -13794.397,E2 -13794.397} C_VEL
LIN {X 0,Y 357.074,Z 522.374,A -85,B 0,C 180,E1 -13796.288,E2 -13796.288} C_VEL
LIN {X 0,Y 359.634,Z 508.005,A -85,B 0,C 180,E1 -13797.972,E2 -13797.972} C_VEL
LIN {X 0,Y 362.23,Z 492.482,A -85,B 0,C 180,E1 -13799.496,E2 -13799.496} C_VEL
LIN {X 0,Y 364.98,Z 475.565,A -85,B 0,C 180,E1 -13800.845,E2 -13800.845} C_VEL
LIN {X 0,Y 366.537,Z 464.791,A -85,B 0,C 180,E1 -13801.568,E2 -13801.568} C_VEL
LIN {X 0,Y 365.628,Z 449.992,A -85,B 0,C 180,E1 -13802.711,E2 -13802.711} C_VEL
LIN {X 0,Y 364.706,Z 435.329,A -85,B 0,C 180,E1 -13803.703,E2 -13803.703} C_VEL
LIN {X 0,Y 362.695,Z 422.613,A -85,B 0,C 180,E1 -13804.621,E2 -13804.621} C_VEL
LIN {X 0,Y 359.955,Z 410.106,A -85,B 0,C 180,E1 -13805.654,E2 -13805.654} C_VEL
LIN {X 0,Y 363.335,Z 399.878,A -85,B 0,C 180,E1 -13808.598,E2 -13808.598} C_VEL
LIN {X 0,Y 364.559,Z 396.789,A -85,B 0,C 180,E1 -13809.546,E2 -13809.546} C_VEL
LIN {X 0,Y 364.834,Z 395.072,A -85,B 0,C 180,E1 -13810.192,E2 -13810.192} C_VEL
LIN {X 0,Y 363.591,Z 390.109,A -85,B 0,C 180,E1 -13812.734,E2 -13812.734} C_VEL
LIN {X 0,Y 362.787,Z 387.842,A -85,B 0,C 180,E1 -13814.221,E2 -13814.221} C_VEL
LIN {X 0,Y 361.486,Z 384.568,A -85,B 0,C 180,E1 -13817.12,E2 -13817.12} C_VEL
LIN {X 0,Y 360.567,Z 382.973,A -85,B 0,C 180,E1 -13819.482,E2 -13819.482} C_VEL
